LIN {X 0,Y 361.915,Z 594.733,A -85,B 0,C 180,E1 -13475.323,E2 -13475.323} C_VEL
LIN {X 0,Y 360.28,Z 612.656,A -85,B 0,C 180,E1 -13478.546,E2 -13478.546} C_VEL
LIN {X 0,Y 358.832,Z 632.276,A -85,B 0,C 180,E1 -13482.004,E2 -13482.004} C_VEL
LIN {X 0,Y 361.379,Z 647.06,A -85,B 0,C 180,E1 -13482.737,E2 -13482.737} C_VEL
LIN {X 0,Y 361.862,Z 654.515,A -85,B 0,C 180,E1 -13483.025,E2 -13483.025} C_VEL
LIN {X 0,Y 359.915,Z 705.535,A -85,B 0,C 180,E1 -13484.534,E2 -13484.534} C_VEL
LIN {X 0,Y 359.371,Z 715.25,A -85,B 0,C 180,E1 -13484.982,E2 -13484.982} C_VEL
LIN {X 0,Y 358.665,Z 725.972,A -85,B 0,C 180,E1 -13485.677,E2 -13485.677} C_VEL
LIN {X 0,Y 357.824,Z 735.392,A -85,B 0,C 180,E1 -13486.512,E2 -13486.512} C_VEL
LIN {X 0,Y 357.037,Z 744.121,A -85,B 0,C 180,E1 -13487.495,E2 -13487.495} C_VEL
LIN {X 0,Y 356.198,Z 752.116,A -85,B 0,C 180,E1 -13488.621,E2 -13488.621} C_VEL
LIN {X 0,Y 355.444,Z 758.493,A -85,B 0,C 180,E1 -13489.75,E2 -13489.75} C_VEL
LIN {X 0,Y 354.734,Z 764.94,A -85,B 0,C 180,E1 -13491.168,E2 -13491.168} C_VEL
LIN {X 0,Y 354.161,Z 770.791,A -85,B 0,C 180,E1 -13492.846,E2 -13492.846} C_VEL
LIN {X 0,Y 353.842,Z 774.432,A -85,B 0,C 180,E1 -13494.301,E2 -13494.301} C_VEL
LIN {X 0,Y 353.51,Z 776.577,A -85,B 0,C 180,E1 -13495.439,E2 -13495.439} C_VEL
LIN {X 0,Y 353.317,Z 778.1,A -85,B 0,C 180,E1 -13496.579,E2 -13496.579} C_VEL
LIN {X 0,Y 353.22,Z 779.024,A -85,B 0,C 180,E1 -13497.719,E2 -13497.719} C_VEL
LIN {X 0,Y 353.166,Z 779.339,A -85,B 0,C 180,E1 -13498.86,E2 -13498.86} C_VEL
LIN {X 0,Y 353.174,Z 779.042,A -85,B 0,C 180,E1 -13500,E2 -13500} C_VEL
LIN {X 0,Y 353.159,Z 778.151,A -85,B 0,C 180,E1 -13501.14,E2 -13501.14} C_VEL
LIN {X 0,Y 353.221,Z 775.737,A -85,B 0,C 180,E1 -13502.851,E2 -13502.851} C_VEL
LIN {X 0,Y 353.366,Z 773.306,A -85,B 0,C 180,E1 -13503.992,E2 -13503.992} C_VEL
LIN {X 0,Y 353.437,Z 770.155,A -85,B 0,C 180,E1 -13505.134,E2 -13505.134} C_VEL
LIN {X 0,Y 353.588,Z 765.013,A -85,B 0,C 180,E1 -13506.57,E2 -13506.57} C_VEL
LIN {X 0,Y 353.957,Z 758.522,A -85,B 0,C 180,E1 -13507.989,E2 -13507.989} C_VEL
LIN {X 0,Y 354.384,Z 750.124,A -85,B 0,C 180,E1 -13509.417,E2 -13509.417} C_VEL
LIN {X 0,Y 354.768,Z 742.674,A -85,B 0,C 180,E1 -13510.415,E2 -13510.415} C_VEL
LIN {X 0,Y 355.307,Z 733.469,A -85,B 0,C 180,E1 -13511.408,E2 -13511.408} C_VEL
LIN {X 0,Y 355.737,Z 722.981,A -85,B 0,C 180,E1 -13512.262,E2 -13512.262} C_VEL
LIN {X 0,Y 356.026,Z 713.566,A -85,B 0,C 180,E1 -13512.831,E2 -13512.831} C_VEL
LIN {X 0,Y 356.368,Z 702.776,A -85,B 0,C 180,E1 -13513.29,E2 -13513.29} C_VEL
LIN {X 0,Y 357.205,Z 650.23,A -85,B 0,C 180,E1 -13514.684,E2 -13514.684} C_VEL
LIN {X 0,Y 355.644,Z 631.764,A -85,B 0,C 180,E1 -13515.249,E2 -13515.249} C_VEL
LIN {X 0,Y 356.547,Z 612.473,A -85,B 0,C 180,E1 -13518.58,E2 -13518.58} C_VEL
LIN {X 0,Y 357.724,Z 591.341,A -85,B 0,C 180,E1 -13522.266,E2 -13522.266} C_VEL
LIN {X 0,Y 359.197,Z 567.38,A -85,B 0,C 180,E1 -13526.454,E2 -13526.454} C_VEL
LIN {X 0,Y 359.427,Z 562.274,A -85,B 0,C 180,E1 -13527.355,E2 -13527.355} C_VEL
LIN {X 0,Y 356.238,Z 546.772,A -85,B 0,C 180,E1 -13530.304,E2 -13530.304} C_VEL
LIN {X 0,Y 354.906,Z 540.412,A -85,B 0,C 180,E1 -13531.563,E2 -13531.563} C_VEL
LIN {X 0,Y 354.817,Z 540.288,A -85,B 0,C 180,E1 -13535.059,E2 -13535.059} C_VEL
LIN {X 0,Y 354.811,Z 540.288,A -85,B 0,C 180,E1 -13537.882,E2 -13537.882} C_VEL
LIN {X 0,Y 354.792,Z 540.268,A -85,B 0,C 180,E1 -13541.171,E2 -13541.171} C_VEL
LIN {X 0,Y 354.795,Z 540.267,A -85,B 0,C 180,E1 -13544.51,E2 -13544.51} C_VEL
LIN {X 0,Y 354.805,Z 540.287,A -85,B 0,C 180,E1 -13547.663,E2 -13547.663} C_VEL
LIN {X 0,Y 354.82,Z 540.262,A -85,B 0,C 180,E1 -13550.666,E2 -13550.666} C_VEL
LIN {X 0,Y 354.826,Z 540.285,A -85,B 0,C 180,E1 -13554.3,E2 -13554.3} C_VEL
LIN {X 0,Y 354.791,Z 540.29,A -85,B 0,C 180,E1 -13557.666,E2 -13557.666} C_VEL
LIN {X 0,Y 354.833,Z 540.286,A -85,B 0,C 180,E1 -13560.632,E2 -13560.632} C_VEL
LIN {X 0,Y 354.938,Z 540.423,A -85,B 0,C 180,E1 -13563.859,E2 -13563.859} C_VEL
LIN {X 0,Y 356.824,Z 549.95,A -85,B 0,C 180,E1 -13566.8,E2 -13566.8} C_VEL
LIN {X 0,Y 357.319,Z 552.539,A -85,B 0,C 180,E1 -13567.484,E2 -13567.484} C_VEL
LIN {X 0,Y 360.175,Z 560.697,A -85,B 0,C 180,E1 -13567.88,E2 -13567.88} C_VEL
LIN {X 0,Y 363.96,Z 579.582,A -85,B 0,C 180,E1 -13568.519,E2 -13568.519} C_VEL
LIN {X 0,Y 362.52,Z 658.642,A -85,B 0,C 180,E1 -13570.093,E2 -13570.093} C_VEL
LIN {X 0,Y 361.977,Z 672.088,A -85,B 0,C 180,E1 -13570.579,E2 -13570.579} C_VEL
LIN {X 0,Y 361.219,Z 684.867,A -85,B 0,C 180,E1 -13571.274,E2 -13571.274} C_VEL
LIN {X 0,Y 360.317,Z 696.201,A -85,B 0,C 180,E1 -13572.108,E2 -13572.108} C_VEL
LIN {X 0,Y 359.181,Z 707.773,A -85,B 0,C 180,E1 -13573.215,E2 -13573.215} C_VEL
LIN {X 0,Y 358.249,Z 718.307,A -85,B 0,C 180,E1 -13574.496,E2 -13574.496} C_VEL
LIN {X 0,Y 357.21,Z 726.851,A -85,B 0,C 180,E1 -13575.762,E2 -13575.762} C_VEL
LIN {X 0,Y 356.22,Z 734.721,A -85,B 0,C 180,E1 -13577.175,E2 -13577.175} C_VEL
LIN {X 0,Y 355.29,Z 742.409,A -85,B 0,C 180,E1 -13578.879,E2 -13578.879} C_VEL
LIN {X 0,Y 354.406,Z 749.468,A -85,B 0,C 180,E1 -13580.871,E2 -13580.871} C_VEL
LIN {X 0,Y 353.946,Z 754.166,A -85,B 0,C 180,E1 -13582.583,E2 -13582.583} C_VEL
LIN {X 0,Y 353.676,Z 757.756,A -85,B 0,C 180,E1 -13584.297,E2 -13584.297} C_VEL
LIN {X 0,Y 353.497,Z 759.613,A -85,B 0,C 180,E1 -13585.438,E2 -13585.438} C_VEL
LIN {X 0,Y 353.34,Z 761.013,A -85,B 0,C 180,E1 -13586.578,E2 -13586.578} C_VEL
LIN {X 0,Y 353.256,Z 762.621,A -85,B 0,C 180,E1 -13588.859,E2 -13588.859} C_VEL
LIN {X 0,Y 353.265,Z 762.853,A -85,B 0,C 180,E1 -13589.999,E2 -13589.999} C_VEL
LIN {X 0,Y 353.256,Z 762.665,A -85,B 0,C 180,E1 -13591.139,E2 -13591.139} C_VEL
LIN {X 0,Y 353.334,Z 761.117,A -85,B 0,C 180,E1 -13593.42,E2 -13593.42} C_VEL
LIN {X 0,Y 353.49,Z 759.761,A -85,B 0,C 180,E1 -13594.56,E2 -13594.56} C_VEL
LIN {X 0,Y 353.814,Z 756.019,A -85,B 0,C 180,E1 -13596.695,E2 -13596.695} C_VEL
LIN {X 0,Y 354.2,Z 751.45,A -85,B 0,C 180,E1 -13598.557,E2 -13598.557} C_VEL
LIN {X 0,Y 355.015,Z 745.015,A -85,B 0,C 180,E1 -13600.55,E2 -13600.55} C_VEL
LIN {X 0,Y 355.811,Z 737.943,A -85,B 0,C 180,E1 -13602.258,E2 -13602.258} C_VEL
LIN {X 0,Y 356.917,Z 729.128,A -85,B 0,C 180,E1 -13603.957,E2 -13603.957} C_VEL
LIN {X 0,Y 358.056,Z 720.077,A -85,B 0,C 180,E1 -13605.365,E2 -13605.365} C_VEL
LIN {X 0,Y 358.248,Z 718.084,A -85,B 0,C 180,E1 -13605.637,E2 -13605.637} C_VEL
LIN {X 0,Y 357.693,Z 714.653,A -85,B 0,C 180,E1 -13606.131,E2 -13606.131} C_VEL
LIN {X 0,Y 353.248,Z 705.711,A -85,B 0,C 180,E1 -13607.436,E2 -13607.436} C_VEL
LIN {X 0,Y 353.002,Z 702.399,A -85,B 0,C 180,E1 -13607.799,E2 -13607.799} C_VEL
LIN {X 0,Y 354.134,Z 690.557,A -85,B 0,C 180,E1 -13608.812,E2 -13608.812} C_VEL
LIN {X 0,Y 355.058,Z 678.47,A -85,B 0,C 180,E1 -13609.587,E2 -13609.587} C_VEL
LIN {X 0,Y 355.635,Z 666.212,A -85,B 0,C 180,E1 -13610.156,E2 -13610.156} C_VEL
LIN {X 0,Y 356.104,Z 654.129,A -85,B 0,C 180,E1 -13610.505,E2 -13610.505} C_VEL
LIN {X 0,Y 357.351,Z 579.83,A -85,B 0,C 180,E1 -13612.003,E2 -13612.003} C_VEL
LIN {X 0,Y 353.421,Z 561.516,A -85,B 0,C 180,E1 -13612.658,E2 -13612.658} C_VEL
LIN {X 0,Y 350.203,Z 552.682,A -85,B 0,C 180,E1 -13613.115,E2 -13613.115} C_VEL
LIN {X 0,Y 348.907,Z 546.369,A -85,B 0,C 180,E1 -13614.983,E2 -13614.983} C_VEL
LIN {X 0,Y 347.866,Z 541.204,A -85,B 0,C 180,E1 -13616.687,E2 -13616.687} C_VEL
LIN {X 0,Y 347.747,Z 541.157,A -85,B 0,C 180,E1 -13620.347,E2 -13620.347} C_VEL
LIN {X 0,Y 347.746,Z 541.17,A -85,B 0,C 180,E1 -13624.043,E2 -13624.043} C_VEL
LIN {X 0,Y 347.763,Z 541.166,A -85,B 0,C 180,E1 -13627.319,E2 -13627.319} C_VEL
LIN {X 0,Y 347.74,Z 541.16,A -85,B 0,C 180,E1 -13630.294,E2 -13630.294} C_VEL
LIN {X 0,Y 347.72,Z 541.166,A -85,B 0,C 180,E1 -13633.407,E2 -13633.407} C_VEL
LIN {X 0,Y 347.742,Z 541.163,A -85,B 0,C 180,E1 -13636.681,E2 -13636.681} C_VEL
LIN {X 0,Y 347.753,Z 541.153,A -85,B 0,C 180,E1 -13640.17,E2 -13640.17} C_VEL
LIN {X 0,Y 347.762,Z 541.151,A -85,B 0,C 180,E1 -13642.679,E2 -13642.679} C_VEL
LIN {X 0,Y 347.757,Z 541.165,A -85,B 0,C 180,E1 -13645.952,E2 -13645.952} C_VEL
LIN {X 0,Y 347.758,Z 541.169,A -85,B 0,C 180,E1 -13649.653,E2 -13649.653} C_VEL
LIN {X 0,Y 347.846,Z 541.145,A -85,B 0,C 180,E1 -13652.744,E2 -13652.744} C_VEL
LIN {X 0,Y 347.782,Z 541.159,A -85,B 0,C 180,E1 -13656.161,E2 -13656.161} C_VEL
LIN {X 0,Y 347.811,Z 541.159,A -85,B 0,C 180,E1 -13659.909,E2 -13659.909} C_VEL
LIN {X 0,Y 347.859,Z 541.147,A -85,B 0,C 180,E1 -13662.359,E2 -13662.359} C_VEL
LIN {X 0,Y 347.89,Z 541.149,A -85,B 0,C 180,E1 -13665.97,E2 -13665.97} C_VEL
LIN {X 0,Y 347.921,Z 541.135,A -85,B 0,C 180,E1 -13669.525,E2 -13669.525} C_VEL
LIN {X 0,Y 348.067,Z 541.126,A -85,B 0,C 180,E1 -13671.874,E2 -13671.874} C_VEL
LIN {X 0,Y 348.06,Z 541.126,A -85,B 0,C 180,E1 -13674.205,E2 -13674.205} C_VEL
LIN {X 0,Y 348.201,Z 541.102,A -85,B 0,C 180,E1 -13677.686,E2 -13677.686} C_VEL
LIN {X 0,Y 348.361,Z 541.091,A -85,B 0,C 180,E1 -13680,E2 -13680} C_VEL
LIN {X 0,Y 348.201,Z 541.103,A -85,B 0,C 180,E1 -13682.313,E2 -13682.313} C_VEL
LIN {X 0,Y 348.101,Z 541.122,A -85,B 0,C 180,E1 -13686.958,E2 -13686.958} C_VEL
LIN {X 0,Y 347.961,Z 541.134,A -85,B 0,C 180,E1 -13689.299,E2 -13689.299} C_VEL
LIN {X 0,Y 347.886,Z 541.148,A -85,B 0,C 180,E1 -13692.84,E2 -13692.84} C_VEL
LIN {X 0,Y 347.832,Z 541.147,A -85,B 0,C 180,E1 -13696.432,E2 -13696.432} C_VEL
LIN {X 0,Y 347.852,Z 541.153,A -85,B 0,C 180,E1 -13698.86,E2 -13698.86} C_VEL
LIN {X 0,Y 347.77,Z 541.159,A -85,B 0,C 180,E1 -13702.58,E2 -13702.58} C_VEL
LIN {X 0,Y 347.806,Z 541.16,A -85,B 0,C 180,E1 -13705.109,E2 -13705.109} C_VEL
LIN {X 0,Y 347.801,Z 541.158,A -85,B 0,C 180,E1 -13707.695,E2 -13707.695} C_VEL
LIN {X 0,Y 347.742,Z 541.163,A -85,B 0,C 180,E1 -13710.349,E2 -13710.349} C_VEL
LIN {X 0,Y 347.742,Z 541.165,A -85,B 0,C 180,E1 -13714.045,E2 -13714.045} C_VEL
LIN {X 0,Y 347.757,Z 541.148,A -85,B 0,C 180,E1 -13717.322,E2 -13717.322} C_VEL
LIN {X 0,Y 347.727,Z 541.169,A -85,B 0,C 180,E1 -13720.298,E2 -13720.298} C_VEL
LIN {X 0,Y 347.742,Z 541.158,A -85,B 0,C 180,E1 -13723.405,E2 -13723.405} C_VEL
LIN {X 0,Y 347.778,Z 541.155,A -85,B 0,C 180,E1 -13726.677,E2 -13726.677} C_VEL
LIN {X 0,Y 347.782,Z 541.157,A -85,B 0,C 180,E1 -13730.166,E2 -13730.166} C_VEL
LIN {X 0,Y 347.786,Z 541.158,A -85,B 0,C 180,E1 -13734.126,E2 -13734.126} C_VEL
LIN {X 0,Y 347.732,Z 541.104,A -85,B 0,C 180,E1 -13738.088,E2 -13738.088} C_VEL
LIN {X 0,Y 347.806,Z 541.332,A -85,B 0,C 180,E1 -13739.197,E2 -13739.197} C_VEL
LIN {X 0,Y 350.44,Z 553.084,A -85,B 0,C 180,E1 -13742.533,E2 -13742.533} C_VEL
LIN {X 0,Y 351.969,Z 561.98,A -85,B 0,C 180,E1 -13744.92,E2 -13744.92} C_VEL
LIN {X 0,Y 351.14,Z 570.572,A -85,B 0,C 180,E1 -13746.977,E2 -13746.977} C_VEL
LIN {X 0,Y 352.793,Z 579.781,A -85,B 0,C 180,E1 -13747.333,E2 -13747.333} C_VEL
LIN {X 0,Y 356.992,Z 605.545,A -85,B 0,C 180,E1 -13748.159,E2 -13748.159} C_VEL
LIN {X 0,Y 355.689,Z 678.841,A -85,B 0,C 180,E1 -13749.659,E2 -13749.659} C_VEL
LIN {X 0,Y 354.909,Z 692.03,A -85,B 0,C 180,E1 -13750.141,E2 -13750.141} C_VEL
LIN {X 0,Y 354.07,Z 704.157,A -85,B 0,C 180,E1 -13750.808,E2 -13750.808} C_VEL
LIN {X 0,Y 352.939,Z 716.406,A -85,B 0,C 180,E1 -13751.723,E2 -13751.723} C_VEL
LIN {X 0,Y 351.697,Z 727.988,A -85,B 0,C 180,E1 -13752.859,E2 -13752.859} C_VEL
LIN {X 0,Y 350.453,Z 738.96,A -85,B 0,C 180,E1 -13754.22,E2 -13754.22} C_VEL
LIN {X 0,Y 349.342,Z 748.628,A -85,B 0,C 180,E1 -13755.734,E2 -13755.734} C_VEL
LIN {X 0,Y 348.199,Z 757.561,A -85,B 0,C 180,E1 -13757.47,E2 -13757.47} C_VEL
LIN {X 0,Y 347.398,Z 764.755,A -85,B 0,C 180,E1 -13759.216,E2 -13759.216} C_VEL
LIN {X 0,Y 346.719,Z 771.306,A -85,B 0,C 180,E1 -13761.257,E2 -13761.257} C_VEL
LIN {X 0,Y 346.343,Z 775.644,A -85,B 0,C 180,E1 -13763.008,E2 -13763.008} C_VEL
LIN {X 0,Y 346.2,Z 777.944,A -85,B 0,C 180,E1 -13764.175,E2 -13764.175} C_VEL
LIN {X 0,Y 346.175,Z 779.809,A -85,B 0,C 180,E1 -13765.343,E2 -13765.343} C_VEL
LIN {X 0,Y 346.147,Z 781.205,A -85,B 0,C 180,E1 -13766.509,E2 -13766.509} C_VEL
LIN {X 0,Y 346.123,Z 784.253,A -85,B 0,C 180,E1 -13770.001,E2 -13770.001} C_VEL
LIN {X 0,Y 346.069,Z 784.599,A -85,B 0,C 180,E1 -13771.165,E2 -13771.165} C_VEL
LIN {X 0,Y 346.081,Z 784.32,A -85,B 0,C 180,E1 -13772.329,E2 -13772.329} C_VEL
LIN {X 0,Y 346.154,Z 783.447,A -85,B 0,C 180,E1 -13773.493,E2 -13773.493} C_VEL
LIN {X 0,Y 346.257,Z 781.07,A -85,B 0,C 180,E1 -13775.242,E2 -13775.242} C_VEL
LIN {X 0,Y 346.431,Z 777.124,A -85,B 0,C 180,E1 -13776.992,E2 -13776.992} C_VEL
LIN {X 0,Y 346.615,Z 773.662,A -85,B 0,C 180,E1 -13778.161,E2 -13778.161} C_VEL
LIN {X 0,Y 347.574,Z 762.458,A -85,B 0,C 180,E1 -13781.371,E2 -13781.371} C_VEL
LIN {X 0,Y 348.549,Z 754.751,A -85,B 0,C 180,E1 -13783.112,E2 -13783.112} C_VEL
LIN {X 0,Y 349.714,Z 745.072,A -85,B 0,C 180,E1 -13784.847,E2 -13784.847} C_VEL
LIN {X 0,Y 350.835,Z 735.09,A -85,B 0,C 180,E1 -13786.288,E2 -13786.288} C_VEL
LIN {X 0,Y 352.096,Z 723.812,A -85,B 0,C 180,E1 -13787.573,E2 -13787.573} C_VEL
LIN {X 0,Y 353.272,Z 712.771,A -85,B 0,C 180,E1 -13788.561,E2 -13788.561} C_VEL
LIN {X 0,Y 354.315,Z 700.533,A -85,B 0,C 180,E1 -13789.406,E2 -13789.406} C_VEL
LIN {X 0,Y 355.211,Z 687.646,A -85,B 0,C 180,E1 -13790.032,E2 -13790.032} C_VEL
LIN {X 0,Y 355.763,Z 673.928,A -85,B 0,C 180,E1 -13790.452,E2 -13790.452} C_VEL
LIN {X 0,Y 356.868,Z 604.856,A -85,B 0,C 180,E1 -13791.849,E2 -13791.849} C_VEL
LIN {X 0,Y 353.3,Z 582.279,A -85,B 0,C 180,E1 -13792.598,E2 -13792.598} C_VEL
LIN {X 0,Y 353.345,Z 575.714,A -85,B 0,C 180,E1 -13793.269,E2 -13793.269} C_VEL
LIN {X 0,Y 352.557,Z 568.23,A -85,B 0,C 180,E1 -13794.231,E2 -13794.231} C_VEL
LIN {X 0,Y 352.055,Z 562.274,A -85,B 0,C 180,E1 -13795.073,E2 -13795.073} C_VEL
LIN {X 0,Y 350.889,Z 555.527,A -85,B 0,C 180,E1 -13796.787,E2 -13796.787} C_VEL
LIN {X 0,Y 348.952,Z 546.205,A -85,B 0,C 180,E1 -13799.368,E2 -13799.368} C_VEL
LIN {X 0,Y 347.804,Z 541.253,A -85,B 0,C 180,E1 -13800.848,E2 -13800.848} C_VEL
LIN {X 0,Y 347.748,Z 541.171,A -85,B 0,C 180,E1 -13804.464,E2 -13804.464} C_VEL
LIN {X 0,Y 347.777,Z 541.167,A -85,B 0,C 180,E1 -13807.989,E2 -13807.989} C_VEL
LIN {X 0,Y 347.755,Z 541.169,A -85,B 0,C 180,E1 -13811.831,E2 -13811.831} C_VEL
LIN {X 0,Y 347.71,Z 541.173,A -85,B 0,C 180,E1 -13815.027,E2 -13815.027} C_VEL
LIN {X 0,Y 347.754,Z 541.168,A -85,B 0,C 180,E1 -13818.398,E2 -13818.398} C_VEL
LIN {X 0,Y 347.821,Z 541.434,A -85,B 0,C 180,E1 -13820.846,E2 -13820.846} C_VEL
LIN {X 0,Y 349.991,Z 546.723,A -85,B 0,C 180,E1 -13822.957,E2 -13822.957} C_VEL
LIN {X 0,Y 352.71,Z 553.567,A -85,B 0,C 180,E1 -13825.28,E2 -13825.28} C_VEL
LIN {X 0,Y 355.393,Z 562,A -85,B 0,C 180,E1 -13827.728,E2 -13827.728} C_VEL
LIN {X 0,Y 357.118,Z 569.16,A -85,B 0,C 180,E1 -13829.556,E2 -13829.556} C_VEL
LIN {X 0,Y 357.945,Z 575.077,A -85,B 0,C 180,E1 -13830.925,E2 -13830.925} C_VEL
LIN {X 0,Y 355.927,Z 592.958,A -85,B 0,C 180,E1 -13834.253,E2 -13834.253} C_VEL
LIN {X 0,Y 353.975,Z 612.503,A -85,B 0,C 180,E1 -13837.837,E2 -13837.837} C_VEL
LIN {X 0,Y 352.348,Z 632.152,A -85,B 0,C 180,E1 -13841.389,E2 -13841.389} C_VEL
LIN {X 0,Y 354.995,Z 647.631,A -85,B 0,C 180,E1 -13842.213,E2 -13842.213} C_VEL
LIN {X 0,Y 355.568,Z 654.786,A -85,B 0,C 180,E1 -13842.508,E2 -13842.508} C_VEL
LIN {X 0,Y 353.443,Z 705.58,A -85,B 0,C 180,E1 -13844.059,E2 -13844.059} C_VEL
LIN {X 0,Y 352.848,Z 715.786,A -85,B 0,C 180,E1 -13844.55,E2 -13844.55} C_VEL
LIN {X 0,Y 352.063,Z 726.264,A -85,B 0,C 180,E1 -13845.255,E2 -13845.255} C_VEL
LIN {X 0,Y 351.177,Z 735.596,A -85,B 0,C 180,E1 -13846.104,E2 -13846.104} C_VEL
LIN {X 0,Y 350.334,Z 744.318,A -85,B 0,C 180,E1 -13847.104,E2 -13847.104} C_VEL
LIN {X 0,Y 349.31,Z 753.123,A -85,B 0,C 180,E1 -13848.393,E2 -13848.393} C_VEL
LIN {X 0,Y 348.519,Z 759.359,A -85,B 0,C 180,E1 -13849.544,E2 -13849.544} C_VEL
LIN {X 0,Y 347.907,Z 764.489,A -85,B 0,C 180,E1 -13850.7,E2 -13850.7} C_VEL
LIN {X 0,Y 347.314,Z 769.751,A -85,B 0,C 180,E1 -13852.179,E2 -13852.179} C_VEL
LIN {X 0,Y 346.981,Z 773.598,A -85,B 0,C 180,E1 -13853.604,E2 -13853.604} C_VEL
LIN {X 0,Y 346.459,Z 776.857,A -85,B 0,C 180,E1 -13855.346,E2 -13855.346} C_VEL
LIN {X 0,Y 346.245,Z 778.294,A -85,B 0,C 180,E1 -13856.509,E2 -13856.509} C_VEL
LIN {X 0,Y 346.131,Z 779.14,A -85,B 0,C 180,E1 -13857.673,E2 -13857.673} C_VEL
LIN {X 0,Y 346.069,Z 779.396,A -85,B 0,C 180,E1 -13858.836,E2 -13858.836} C_VEL
LIN {X 0,Y 346.075,Z 779.038,A -85,B 0,C 180,E1 -13860,E2 -13860} C_VEL
LIN {X 0,Y 346.062,Z 778.065,A -85,B 0,C 180,E1 -13861.164,E2 -13861.164} C_VEL
LIN {X 0,Y 346.142,Z 775.463,A -85,B 0,C 180,E1 -13862.91,E2 -13862.91} C_VEL
LIN {X 0,Y 346.327,Z 771.383,A -85,B 0,C 180,E1 -13864.656,E2 -13864.656} C_VEL
LIN {X 0,Y 346.451,Z 766.163,A -85,B 0,C 180,E1 -13866.274,E2 -13866.274} C_VEL
LIN {X 0,Y 346.772,Z 760.656,A -85,B 0,C 180,E1 -13867.57,E2 -13867.57} C_VEL
LIN {X 0,Y 347.053,Z 754.557,A -85,B 0,C 180,E1 -13868.736,E2 -13868.736} C_VEL
LIN {X 0,Y 347.516,Z 747.094,A -85,B 0,C 180,E1 -13869.898,E2 -13869.898} C_VEL
LIN {X 0,Y 347.944,Z 737.609,A -85,B 0,C 180,E1 -13871.063,E2 -13871.063} C_VEL
LIN {X 0,Y 348.344,Z 730.147,A -85,B 0,C 180,E1 -13871.787,E2 -13871.787} C_VEL
LIN {X 0,Y 348.734,Z 720.716,A -85,B 0,C 180,E1 -13872.512,E2 -13872.512} C_VEL
LIN {X 0,Y 349.065,Z 709.842,A -85,B 0,C 180,E1 -13873.129,E2 -13873.129} C_VEL
LIN {X 0,Y 349.317,Z 698.696,A -85,B 0,C 180,E1 -13873.526,E2 -13873.526} C_VEL
LIN {X 0,Y 350.173,Z 650.419,A -85,B 0,C 180,E1 -13874.836,E2 -13874.836} C_VEL
LIN {X 0,Y 348.579,Z 631.804,A -85,B 0,C 180,E1 -13875.42,E2 -13875.42} C_VEL
LIN {X 0,Y 349.497,Z 614.378,A -85,B 0,C 180,E1 -13878.465,E2 -13878.465} C_VEL
LIN {X 0,Y 350.718,Z 592.221,A -85,B 0,C 180,E1 -13882.38,E2 -13882.38} C_VEL
LIN {X 0,Y 352.133,Z 569.733,A -85,B 0,C 180,E1 -13886.364,E2 -13886.364} C_VEL
LIN {X 0,Y 352.366,Z 562.799,A -85,B 0,C 180,E1 -13887.606,E2 -13887.606} C_VEL
LIN {X 0,Y 348.783,Z 545.615,A -85,B 0,C 180,E1 -13890.919,E2 -13890.919} C_VEL
LIN {X 0,Y 347.831,Z 541.279,A -85,B 0,C 180,E1 -13891.824,E2 -13891.824} C_VEL
LIN {X 0,Y 347.775,Z 541.166,A -85,B 0,C 180,E1 -13896.065,E2 -13896.065} C_VEL
LIN {X 0,Y 347.757,Z 541.165,A -85,B 0,C 180,E1 -13898.792,E2 -13898.792} C_VEL
LIN {X 0,Y 347.755,Z 541.134,A -85,B 0,C 180,E1 -13901.83,E2 -13901.83} C_VEL
LIN {X 0,Y 347.773,Z 541.149,A -85,B 0,C 180,E1 -13905.016,E2 -13905.016} C_VEL
LIN {X 0,Y 347.758,Z 541.158,A -85,B 0,C 180,E1 -13908.396,E2 -13908.396} C_VEL
LIN {X 0,Y 347.778,Z 541.153,A -85,B 0,C 180,E1 -13912.011,E2 -13912.011} C_VEL
LIN {X 0,Y 347.749,Z 541.156,A -85,B 0,C 180,E1 -13915.536,E2 -13915.536} C_VEL
LIN {X 0,Y 347.765,Z 541.165,A -85,B 0,C 180,E1 -13919.653,E2 -13919.653} C_VEL
LIN {X 0,Y 347.898,Z 541.272,A -85,B 0,C 180,E1 -13923.48,E2 -13923.48} C_VEL
LIN {X 0,Y 349.965,Z 551.705,A -85,B 0,C 180,E1 -13926.765,E2 -13926.765} C_VEL
LIN {X 0,Y 350.215,Z 552.95,A -85,B 0,C 180,E1 -13927.018,E2 -13927.018} C_VEL
LIN {X 0,Y 353.926,Z 563.384,A -85,B 0,C 180,E1 -13927.522,E2 -13927.522} C_VEL
LIN {X 0,Y 357.365,Z 580.665,A -85,B 0,C 180,E1 -13928.12,E2 -13928.12} C_VEL
LIN {X 0,Y 355.876,Z 658.864,A -85,B 0,C 180,E1 -13929.705,E2 -13929.705} C_VEL
LIN {X 0,Y 355.298,Z 672.303,A -85,B 0,C 180,E1 -13930.199,E2 -13930.199} C_VEL
LIN {X 0,Y 354.52,Z 685.079,A -85,B 0,C 180,E1 -13930.907,E2 -13930.907} C_VEL
LIN {X 0,Y 353.585,Z 696.411,A -85,B 0,C 180,E1 -13931.756,E2 -13931.756} C_VEL
LIN {X 0,Y 352.511,Z 706.905,A -85,B 0,C 180,E1 -13932.763,E2 -13932.763} C_VEL
LIN {X 0,Y 351.509,Z 717.451,A -85,B 0,C 180,E1 -13934.042,E2 -13934.042} C_VEL
LIN {X 0,Y 350.339,Z 727.058,A -85,B 0,C 180,E1 -13935.477,E2 -13935.477} C_VEL
LIN {X 0,Y 349.282,Z 734.929,A -85,B 0,C 180,E1 -13936.916,E2 -13936.916} C_VEL
LIN {X 0,Y 348.321,Z 742.616,A -85,B 0,C 180,E1 -13938.654,E2 -13938.654} C_VEL
LIN {X 0,Y 347.656,Z 747.864,A -85,B 0,C 180,E1 -13940.105,E2 -13940.105} C_VEL
LIN {X 0,Y 347.019,Z 752.957,A -85,B 0,C 180,E1 -13941.849,E2 -13941.849} C_VEL
LIN {X 0,Y 346.728,Z 756.326,A -85,B 0,C 180,E1 -13943.32,E2 -13943.32} C_VEL
LIN {X 0,Y 346.439,Z 759.818,A -85,B 0,C 180,E1 -13945.345,E2 -13945.345} C_VEL
LIN {X 0,Y 346.264,Z 761.218,A -85,B 0,C 180,E1 -13946.508,E2 -13946.508} C_VEL
LIN {X 0,Y 346.16,Z 762.826,A -85,B 0,C 180,E1 -13948.836,E2 -13948.836} C_VEL
LIN {X 0,Y 346.168,Z 763.058,A -85,B 0,C 180,E1 -13949.999,E2 -13949.999} C_VEL
LIN {X 0,Y 346.159,Z 762.869,A -85,B 0,C 180,E1 -13951.162,E2 -13951.162} C_VEL
LIN {X 0,Y 346.259,Z 761.321,A -85,B 0,C 180,E1 -13953.49,E2 -13953.49} C_VEL
LIN {X 0,Y 346.432,Z 759.964,A -85,B 0,C 180,E1 -13954.653,E2 -13954.653} C_VEL
LIN {X 0,Y 346.727,Z 756.547,A -85,B 0,C 180,E1 -13956.679,E2 -13956.679} C_VEL
LIN {X 0,Y 347.175,Z 751.654,A -85,B 0,C 180,E1 -13958.732,E2 -13958.732} C_VEL
LIN {X 0,Y 348.004,Z 745.219,A -85,B 0,C 180,E1 -13960.765,E2 -13960.765} C_VEL
LIN {X 0,Y 348.861,Z 738.146,A -85,B 0,C 180,E1 -13962.506,E2 -13962.506} C_VEL
LIN {X 0,Y 350.045,Z 729.329,A -85,B 0,C 180,E1 -13964.237,E2 -13964.237} C_VEL
LIN {X 0,Y 351.213,Z 720.288,A -85,B 0,C 180,E1 -13965.67,E2 -13965.67} C_VEL
LIN {X 0,Y 352.302,Z 709.234,A -85,B 0,C 180,E1 -13967.081,E2 -13967.081} C_VEL
LIN {X 0,Y 353.002,Z 702.399,A -85,B 0,C 180,E1 -13967.799,E2 -13967.799} C_VEL
LIN {X 0,Y 352.983,Z 697.369,A -85,B 0,C 180,E1 -13968.302,E2 -13968.302} C_VEL
LIN {X 0,Y 351.028,Z 689.052,A -85,B 0,C 180,E1 -13969.125,E2 -13969.125} C_VEL
LIN {X 0,Y 348.89,Z 680.413,A -85,B 0,C 180,E1 -13969.847,E2 -13969.847} C_VEL
LIN {X 0,Y 348.576,Z 674.878,A -85,B 0,C 180,E1 -13970.184,E2 -13970.184} C_VEL
LIN {X 0,Y 349.199,Z 663.426,A -85,B 0,C 180,E1 -13970.66,E2 -13970.66} C_VEL
LIN {X 0,Y 349.622,Z 645.492,A -85,B 0,C 180,E1 -13971.096,E2 -13971.096} C_VEL
LIN {X 0,Y 350.73,Z 580.722,A -85,B 0,C 180,E1 -13972.426,E2 -13972.426} C_VEL
LIN {X 0,Y 347.06,Z 563.542,A -85,B 0,C 180,E1 -13973.057,E2 -13973.057} C_VEL
LIN {X 0,Y 343.049,Z 552.944,A -85,B 0,C 180,E1 -13973.62,E2 -13973.62} C_VEL
LIN {X 0,Y 341.508,Z 545.362,A -85,B 0,C 180,E1 -13975.931,E2 -13975.931} C_VEL
LIN {X 0,Y 340.834,Z 542.049,A -85,B 0,C 180,E1 -13977.111,E2 -13977.111} C_VEL
LIN {X 0,Y 340.696,Z 542.044,A -85,B 0,C 180,E1 -13981.043,E2 -13981.043} C_VEL
LIN {X 0,Y 340.716,Z 542.04,A -85,B 0,C 180,E1 -13985.277,E2 -13985.277} C_VEL
LIN {X 0,Y 340.71,Z 542.043,A -85,B 0,C 180,E1 -13988.386,E2 -13988.386} C_VEL
LIN {X 0,Y 340.699,Z 542.046,A -85,B 0,C 180,E1 -13992.045,E2 -13992.045} C_VEL
LIN {X 0,Y 340.663,Z 542.045,A -85,B 0,C 180,E1 -13996.223,E2 -13996.223} C_VEL
LIN {X 0,Y 340.7,Z 542.044,A -85,B 0,C 180,E1 -13998.692,E2 -13998.692} C_VEL
LIN {X 0,Y 340.736,Z 542.019,A -85,B 0,C 180,E1 -14001.773,E2 -14001.773} C_VEL
LIN {X 0,Y 340.727,Z 542.044,A -85,B 0,C 180,E1 -14005.592,E2 -14005.592} C_VEL
LIN {X 0,Y 340.757,Z 542.038,A -85,B 0,C 180,E1 -14010.021,E2 -14010.021} C_VEL
LIN {X 0,Y 340.799,Z 542.024,A -85,B 0,C 180,E1 -14013.019,E2 -14013.019} C_VEL
LIN {X 0,Y 340.722,Z 542.039,A -85,B 0,C 180,E1 -14016.927,E2 -14016.927} C_VEL
LIN {X 0,Y 340.788,Z 542.032,A -85,B 0,C 180,E1 -14020.733,E2 -14020.733} C_VEL
LIN {X 0,Y 340.779,Z 542.026,A -85,B 0,C 180,E1 -14023.218,E2 -14023.218} C_VEL
LIN {X 0,Y 340.837,Z 542.027,A -85,B 0,C 180,E1 -14026.89,E2 -14026.89} C_VEL
LIN {X 0,Y 340.921,Z 542.004,A -85,B 0,C 180,E1 -14030.507,E2 -14030.507} C_VEL
LIN {X 0,Y 341.068,Z 541.997,A -85,B 0,C 180,E1 -14032.898,E2 -14032.898} C_VEL
LIN {X 0,Y 341.163,Z 541.977,A -85,B 0,C 180,E1 -14037.639,E2 -14037.639} C_VEL
LIN {X 0,Y 341.31,Z 541.97,A -85,B 0,C 180,E1 -14040,E2 -14040} C_VEL
LIN {X 0,Y 341.163,Z 541.979,A -85,B 0,C 180,E1 -14042.361,E2 -14042.361} C_VEL
LIN {X 0,Y 341.07,Z 541.999,A -85,B 0,C 180,E1 -14047.102,E2 -14047.102} C_VEL
LIN {X 0,Y 340.866,Z 542.013,A -85,B 0,C 180,E1 -14050.694,E2 -14050.694} C_VEL
LIN {X 0,Y 340.855,Z 542.022,A -85,B 0,C 180,E1 -14054.325,E2 -14054.325} C_VEL
LIN {X 0,Y 340.831,Z 542.027,A -85,B 0,C 180,E1 -14058.468,E2 -14058.468} C_VEL
LIN {X 0,Y 340.746,Z 542.033,A -85,B 0,C 180,E1 -14061.857,E2 -14061.857} C_VEL
LIN {X 0,Y 340.765,Z 542.034,A -85,B 0,C 180,E1 -14065.665,E2 -14065.665} C_VEL
LIN {X 0,Y 340.721,Z 542.042,A -85,B 0,C 180,E1 -14068.321,E2 -14068.321} C_VEL
LIN {X 0,Y 340.691,Z 542.041,A -85,B 0,C 180,E1 -14071.045,E2 -14071.045} C_VEL
LIN {X 0,Y 340.712,Z 542.032,A -85,B 0,C 180,E1 -14075.28,E2 -14075.28} C_VEL
LIN {X 0,Y 340.705,Z 542.042,A -85,B 0,C 180,E1 -14078.387,E2 -14078.387} C_VEL
LIN {X 0,Y 340.696,Z 542.032,A -85,B 0,C 180,E1 -14082.047,E2 -14082.047} C_VEL
LIN {X 0,Y 340.731,Z 542.043,A -85,B 0,C 180,E1 -14085.471,E2 -14085.471} C_VEL
LIN {X 0,Y 340.721,Z 542.043,A -85,B 0,C 180,E1 -14088.697,E2 -14088.697} C_VEL
LIN {X 0,Y 340.735,Z 542.013,A -85,B 0,C 180,E1 -14091.775,E2 -14091.775} C_VEL
LIN {X 0,Y 340.72,Z 542.037,A -85,B 0,C 180,E1 -14095.596,E2 -14095.596} C_VEL
LIN {X 0,Y 340.735,Z 542.067,A -85,B 0,C 180,E1 -14098.702,E2 -14098.702} C_VEL
LIN {X 0,Y 343.178,Z 552.874,A -85,B 0,C 180,E1 -14101.901,E2 -14101.901} C_VEL
LIN {X 0,Y 345.004,Z 562.916,A -85,B 0,C 180,E1 -14104.674,E2 -14104.674} C_VEL
LIN {X 0,Y 344.445,Z 569.181,A -85,B 0,C 180,E1 -14106.252,E2 -14106.252} C_VEL
LIN {X 0,Y 344.392,Z 570.812,A -85,B 0,C 180,E1 -14106.533,E2 -14106.533} C_VEL
LIN {X 0,Y 349.428,Z 599.924,A -85,B 0,C 180,E1 -14107.543,E2 -14107.543} C_VEL
LIN {X 0,Y 350.388,Z 608.082,A -85,B 0,C 180,E1 -14107.784,E2 -14107.784} C_VEL
LIN {X 0,Y 349.044,Z 678.649,A -85,B 0,C 180,E1 -14109.254,E2 -14109.254} C_VEL
LIN {X 0,Y 348.247,Z 691.834,A -85,B 0,C 180,E1 -14109.744,E2 -14109.744} C_VEL
LIN {X 0,Y 347.369,Z 703.959,A -85,B 0,C 180,E1 -14110.423,E2 -14110.423} C_VEL
LIN {X 0,Y 346.199,Z 716.206,A -85,B 0,C 180,E1 -14111.354,E2 -14111.354} C_VEL
LIN {X 0,Y 344.91,Z 727.787,A -85,B 0,C 180,E1 -14112.511,E2 -14112.511} C_VEL
LIN {X 0,Y 343.683,Z 737.768,A -85,B 0,C 180,E1 -14113.76,E2 -14113.76} C_VEL
LIN {X 0,Y 342.61,Z 746.748,A -85,B 0,C 180,E1 -14115.144,E2 -14115.144} C_VEL
LIN {X 0,Y 341.623,Z 754.621,A -85,B 0,C 180,E1 -14116.619,E2 -14116.619} C_VEL
LIN {X 0,Y 340.578,Z 762.31,A -85,B 0,C 180,E1 -14118.394,E2 -14118.394} C_VEL
LIN {X 0,Y 340.035,Z 767.584,A -85,B 0,C 180,E1 -14119.883,E2 -14119.883} C_VEL
LIN {X 0,Y 339.53,Z 772.693,A -85,B 0,C 180,E1 -14121.67,E2 -14121.67} C_VEL
LIN {X 0,Y 339.175,Z 776.666,A -85,B 0,C 180,E1 -14123.457,E2 -14123.457} C_VEL
LIN {X 0,Y 339.076,Z 779.604,A -85,B 0,C 180,E1 -14125.245,E2 -14125.245} C_VEL
LIN {X 0,Y 339.071,Z 781.001,A -85,B 0,C 180,E1 -14126.436,E2 -14126.436} C_VEL
LIN {X 0,Y 339.025,Z 784.082,A -85,B 0,C 180,E1 -14130.001,E2 -14130.001} C_VEL
LIN {X 0,Y 338.974,Z 784.495,A -85,B 0,C 180,E1 -14131.189,E2 -14131.189} C_VEL
LIN {X 0,Y 338.996,Z 784.308,A -85,B 0,C 180,E1 -14132.377,E2 -14132.377} C_VEL
LIN {X 0,Y 339.083,Z 783.534,A -85,B 0,C 180,E1 -14133.566,E2 -14133.566} C_VEL
LIN {X 0,Y 339.174,Z 782.165,A -85,B 0,C 180,E1 -14134.755,E2 -14134.755} C_VEL
LIN {X 0,Y 339.291,Z 778.97,A -85,B 0,C 180,E1 -14136.542,E2 -14136.542} C_VEL
LIN {X 0,Y 339.61,Z 774.18,A -85,B 0,C 180,E1 -14138.33,E2 -14138.33} C_VEL
LIN {X 0,Y 339.93,Z 768.846,A -85,B 0,C 180,E1 -14139.822,E2 -14139.822} C_VEL
LIN {X 0,Y 341.062,Z 758.612,A -85,B 0,C 180,E1 -14142.497,E2 -14142.497} C_VEL
LIN {X 0,Y 342.187,Z 749.97,A -85,B 0,C 180,E1 -14144.269,E2 -14144.269} C_VEL
LIN {X 0,Y 343.301,Z 740.669,A -85,B 0,C 180,E1 -14145.808,E2 -14145.808} C_VEL
LIN {X 0,Y 344.548,Z 730.205,A -85,B 0,C 180,E1 -14147.204,E2 -14147.204} C_VEL
LIN {X 0,Y 345.832,Z 719.197,A -85,B 0,C 180,E1 -14148.361,E2 -14148.361} C_VEL
LIN {X 0,Y 347.086,Z 706.87,A -85,B 0,C 180,E1 -14149.365,E2 -14149.365} C_VEL
LIN {X 0,Y 348.003,Z 695.188,A -85,B 0,C 180,E1 -14150.08,E2 -14150.08} C_VEL
LIN {X 0,Y 348.843,Z 682.703,A -85,B 0,C 180,E1 -14150.607,E2 -14150.607} C_VEL
LIN {X 0,Y 349.29,Z 666.77,A -85,B 0,C 180,E1 -14151.003,E2 -14151.003} C_VEL
LIN {X 0,Y 350.262,Z 605.856,A -85,B 0,C 180,E1 -14152.257,E2 -14152.257} C_VEL
LIN {X 0,Y 347.594,Z 588.463,A -85,B 0,C 180,E1 -14152.831,E2 -14152.831} C_VEL
LIN {X 0,Y 347.893,Z 578.676,A -85,B 0,C 180,E1 -14153.831,E2 -14153.831} C_VEL
LIN {X 0,Y 347.302,Z 571.517,A -85,B 0,C 180,E1 -14154.797,E2 -14154.797} C_VEL
LIN {X 0,Y 346.827,Z 565.788,A -85,B 0,C 180,E1 -14155.625,E2 -14155.625} C_VEL
LIN {X 0,Y 343.781,Z 554.509,A -85,B 0,C 180,E1 -14158.048,E2 -14158.048} C_VEL
LIN {X 0,Y 341.81,Z 546.171,A -85,B 0,C 180,E1 -14160.28,E2 -14160.28} C_VEL
LIN {X 0,Y 340.953,Z 543.1,A -85,B 0,C 180,E1 -14161.365,E2 -14161.365} C_VEL
LIN {X 0,Y 340.743,Z 542.208,A -85,B 0,C 180,E1 -14161.86,E2 -14161.86} C_VEL
LIN {X 0,Y 340.722,Z 542.041,A -85,B 0,C 180,E1 -14165.279,E2 -14165.279} C_VEL
LIN {X 0,Y 340.713,Z 542.043,A -85,B 0,C 180,E1 -14168.387,E2 -14168.387} C_VEL
LIN {X 0,Y 340.703,Z 542.045,A -85,B 0,C 180,E1 -14172.046,E2 -14172.046} C_VEL
LIN {X 0,Y 340.656,Z 542.05,A -85,B 0,C 180,E1 -14176.227,E2 -14176.227} C_VEL
LIN {X 0,Y 340.746,Z 542.217,A -85,B 0,C 180,E1 -14178.607,E2 -14178.607} C_VEL
LIN {X 0,Y 341.338,Z 544.229,A -85,B 0,C 180,E1 -14179.625,E2 -14179.625} C_VEL
LIN {X 0,Y 342.329,Z 545.699,A -85,B 0,C 180,E1 -14180.474,E2 -14180.474} C_VEL
LIN {X 0,Y 345.085,Z 552.234,A -85,B 0,C 180,E1 -14183.18,E2 -14183.18} C_VEL
LIN {X 0,Y 347.569,Z 559.075,A -85,B 0,C 180,E1 -14185.516,E2 -14185.516} C_VEL
LIN {X 0,Y 350.173,Z 568.166,A -85,B 0,C 180,E1 -14188.165,E2 -14188.165} C_VEL
LIN {X 0,Y 351.589,Z 575.463,A -85,B 0,C 180,E1 -14190.018,E2 -14190.018} C_VEL
LIN {X 0,Y 351.765,Z 578.502,A -85,B 0,C 180,E1 -14190.693,E2 -14190.693} C_VEL
LIN {X 0,Y 349.163,Z 599.541,A -85,B 0,C 180,E1 -14194.677,E2 -14194.677} C_VEL
LIN {X 0,Y 346.961,Z 620.579,A -85,B 0,C 180,E1 -14198.617,E2 -14198.617} C_VEL
LIN {X 0,Y 345.971,Z 632.069,A -85,B 0,C 180,E1 -14200.725,E2 -14200.725} C_VEL
LIN {X 0,Y 348.648,Z 647.472,A -85,B 0,C 180,E1 -14201.605,E2 -14201.605} C_VEL
LIN {X 0,Y 349.329,Z 655.763,A -85,B 0,C 180,E1 -14201.975,E2 -14201.975} C_VEL
LIN {X 0,Y 347.034,Z 705.884,A -85,B 0,C 180,E1 -14203.567,E2 -14203.567} C_VEL
LIN {X 0,Y 346.345,Z 716.637,A -85,B 0,C 180,E1 -14204.101,E2 -14204.101} C_VEL
LIN {X 0,Y 345.507,Z 726.85,A -85,B 0,C 180,E1 -14204.818,E2 -14204.818} C_VEL
LIN {X 0,Y 344.565,Z 736.061,A -85,B 0,C 180,E1 -14205.682,E2 -14205.682} C_VEL
LIN {X 0,Y 343.656,Z 744.655,A -85,B 0,C 180,E1 -14206.699,E2 -14206.699} C_VEL
LIN {X 0,Y 342.692,Z 752.507,A -85,B 0,C 180,E1 -14207.865,E2 -14207.865} C_VEL
LIN {X 0,Y 341.838,Z 758.831,A -85,B 0,C 180,E1 -14209.037,E2 -14209.037} C_VEL
LIN {X 0,Y 340.961,Z 765.248,A -85,B 0,C 180,E1 -14210.509,E2 -14210.509} C_VEL
LIN {X 0,Y 340.438,Z 769.342,A -85,B 0,C 180,E1 -14211.691,E2 -14211.691} C_VEL
LIN {X 0,Y 339.99,Z 773.575,A -85,B 0,C 180,E1 -14213.248,E2 -14213.248} C_VEL
LIN {X 0,Y 339.412,Z 777.167,A -85,B 0,C 180,E1 -14215.249,E2 -14215.249} C_VEL
LIN {X 0,Y 339.175,Z 778.501,A -85,B 0,C 180,E1 -14216.436,E2 -14216.436} C_VEL
LIN {X 0,Y 339.046,Z 779.248,A -85,B 0,C 180,E1 -14217.624,E2 -14217.624} C_VEL
LIN {X 0,Y 338.976,Z 779.418,A -85,B 0,C 180,E1 -14218.812,E2 -14218.812} C_VEL
LIN {X 0,Y 338.978,Z 778.994,A -85,B 0,C 180,E1 -14220,E2 -14220} C_VEL
LIN {X 0,Y 338.969,Z 777.954,A -85,B 0,C 180,E1 -14221.188,E2 -14221.188} C_VEL
LIN {X 0,Y 339.065,Z 775.17,A -85,B 0,C 180,E1 -14222.97,E2 -14222.97} C_VEL
LIN {X 0,Y 339.245,Z 770.96,A -85,B 0,C 180,E1 -14224.753,E2 -14224.753} C_VEL
LIN {X 0,Y 339.342,Z 766.238,A -85,B 0,C 180,E1 -14226.215,E2 -14226.215} C_VEL
LIN {X 0,Y 339.707,Z 759.815,A -85,B 0,C 180,E1 -14227.728,E2 -14227.728} C_VEL
LIN {X 0,Y 340.033,Z 753.543,A -85,B 0,C 180,E1 -14228.918,E2 -14228.918} C_VEL
LIN {X 0,Y 340.433,Z 744.725,A -85,B 0,C 180,E1 -14230.257,E2 -14230.257} C_VEL
LIN {X 0,Y 340.973,Z 735.921,A -85,B 0,C 180,E1 -14231.292,E2 -14231.292} C_VEL
LIN {X 0,Y 341.41,Z 726.404,A -85,B 0,C 180,E1 -14232.181,E2 -14232.181} C_VEL
LIN {X 0,Y 341.811,Z 715.597,A -85,B 0,C 180,E1 -14232.921,E2 -14232.921} C_VEL
LIN {X 0,Y 342.162,Z 705.694,A -85,B 0,C 180,E1 -14233.398,E2 -14233.398} C_VEL
LIN {X 0,Y 342.695,Z 680.967,A -85,B 0,C 180,E1 -14234.133,E2 -14234.133} C_VEL
LIN {X 0,Y 343.124,Z 650.323,A -85,B 0,C 180,E1 -14235.002,E2 -14235.002} C_VEL
LIN {X 0,Y 341.549,Z 631.796,A -85,B 0,C 180,E1 -14235.592,E2 -14235.592} C_VEL
LIN {X 0,Y 342.487,Z 613.426,A -85,B 0,C 180,E1 -14238.857,E2 -14238.857} C_VEL
LIN {X 0,Y 343.73,Z 592.833,A -85,B 0,C 180,E1 -14242.543,E2 -14242.543} C_VEL
LIN {X 0,Y 345.211,Z 570.176,A -85,B 0,C 180,E1 -14246.608,E2 -14246.608} C_VEL
LIN {X 0,Y 345.468,Z 564.872,A -85,B 0,C 180,E1 -14247.569,E2 -14247.569} C_VEL
LIN {X 0,Y 342.671,Z 551.016,A -85,B 0,C 180,E1 -14250.261,E2 -14250.261} C_VEL
LIN {X 0,Y 340.776,Z 542.168,A -85,B 0,C 180,E1 -14252.068,E2 -14252.068} C_VEL
LIN {X 0,Y 340.723,Z 542.043,A -85,B 0,C 180,E1 -14255.279,E2 -14255.279} C_VEL
LIN {X 0,Y 340.715,Z 542.047,A -85,B 0,C 180,E1 -14258.386,E2 -14258.386} C_VEL
LIN {X 0,Y 340.703,Z 542.008,A -85,B 0,C 180,E1 -14262.045,E2 -14262.045} C_VEL
LIN {X 0,Y 340.702,Z 542.039,A -85,B 0,C 180,E1 -14265.463,E2 -14265.463} C_VEL
LIN {X 0,Y 340.693,Z 542.034,A -85,B 0,C 180,E1 -14268.69,E2 -14268.69} C_VEL
LIN {X 0,Y 340.737,Z 542.026,A -85,B 0,C 180,E1 -14271.772,E2 -14271.772} C_VEL
LIN {X 0,Y 340.727,Z 542.031,A -85,B 0,C 180,E1 -14275.595,E2 -14275.595} C_VEL
LIN {X 0,Y 340.773,Z 542.038,A -85,B 0,C 180,E1 -14280.02,E2 -14280.02} C_VEL
LIN {X 0,Y 340.848,Z 542.17,A -85,B 0,C 180,E1 -14283.106,E2 -14283.106} C_VEL
LIN {X 0,Y 342.923,Z 552.514,A -85,B 0,C 180,E1 -14286.407,E2 -14286.407} C_VEL
LIN {X 0,Y 343.308,Z 553.925,A -85,B 0,C 180,E1 -14286.557,E2 -14286.557} C_VEL
LIN {X 0,Y 347.609,Z 565.502,A -85,B 0,C 180,E1 -14287.132,E2 -14287.132} C_VEL
LIN {X 0,Y 350.817,Z 581.563,A -85,B 0,C 180,E1 -14287.704,E2 -14287.704} C_VEL
LIN {X 0,Y 349.24,Z 659.086,A -85,B 0,C 180,E1 -14289.302,E2 -14289.302} C_VEL
LIN {X 0,Y 348.636,Z 672.518,A -85,B 0,C 180,E1 -14289.804,E2 -14289.804} C_VEL
LIN {X 0,Y 347.845,Z 685.291,A -85,B 0,C 180,E1 -14290.525,E2 -14290.525} C_VEL
LIN {X 0,Y 346.855,Z 696.621,A -85,B 0,C 180,E1 -14291.389,E2 -14291.389} C_VEL
LIN {X 0,Y 345.73,Z 707.114,A -85,B 0,C 180,E1 -14292.414,E2 -14292.414} C_VEL
LIN {X 0,Y 344.672,Z 717.723,A -85,B 0,C 180,E1 -14293.726,E2 -14293.726} C_VEL
LIN {X 0,Y 343.472,Z 727.266,A -85,B 0,C 180,E1 -14295.18,E2 -14295.18} C_VEL
LIN {X 0,Y 342.372,Z 735.136,A -85,B 0,C 180,E1 -14296.647,E2 -14296.647} C_VEL
LIN {X 0,Y 341.341,Z 742.823,A -85,B 0,C 180,E1 -14298.418,E2 -14298.418} C_VEL
LIN {X 0,Y 340.658,Z 748.071,A -85,B 0,C 180,E1 -14299.899,E2 -14299.899} C_VEL
LIN {X 0,Y 339.994,Z 753.163,A -85,B 0,C 180,E1 -14301.679,E2 -14301.679} C_VEL
LIN {X 0,Y 339.638,Z 756.863,A -85,B 0,C 180,E1 -14303.34,E2 -14303.34} C_VEL
LIN {X 0,Y 339.383,Z 760.023,A -85,B 0,C 180,E1 -14305.248,E2 -14305.248} C_VEL
LIN {X 0,Y 339.192,Z 761.423,A -85,B 0,C 180,E1 -14306.435,E2 -14306.435} C_VEL
LIN {X 0,Y 339.063,Z 763.031,A -85,B 0,C 180,E1 -14308.811,E2 -14308.811} C_VEL
LIN {X 0,Y 339.072,Z 763.263,A -85,B 0,C 180,E1 -14309.999,E2 -14309.999} C_VEL
LIN {X 0,Y 339.062,Z 763.074,A -85,B 0,C 180,E1 -14311.187,E2 -14311.187} C_VEL
LIN {X 0,Y 339.187,Z 761.525,A -85,B 0,C 180,E1 -14313.563,E2 -14313.563} C_VEL
LIN {X 0,Y 339.376,Z 760.168,A -85,B 0,C 180,E1 -14314.75,E2 -14314.75} C_VEL
LIN {X 0,Y 339.634,Z 757.082,A -85,B 0,C 180,E1 -14316.655,E2 -14316.655} C_VEL
LIN {X 0,Y 339.991,Z 753.414,A -85,B 0,C 180,E1 -14318.319,E2 -14318.319} C_VEL
LIN {X 0,Y 340.632,Z 748.4,A -85,B 0,C 180,E1 -14320.099,E2 -14320.099} C_VEL
LIN {X 0,Y 341.435,Z 742.087,A -85,B 0,C 180,E1 -14321.877,E2 -14321.877} C_VEL
LIN {X 0,Y 342.457,Z 734.181,A -85,B 0,C 180,E1 -14323.65,E2 -14323.65} C_VEL
LIN {X 0,Y 343.909,Z 724.341,A -85,B 0,C 180,E1 -14325.405,E2 -14325.405} C_VEL
LIN {X 0,Y 345.033,Z 714.022,A -85,B 0,C 180,E1 -14326.872,E2 -14326.872} C_VEL
LIN {X 0,Y 346.216,Z 702.824,A -85,B 0,C 180,E1 -14328.136,E2 -14328.136} C_VEL
LIN {X 0,Y 347.42,Z 690.754,A -85,B 0,C 180,E1 -14329.19,E2 -14329.19} C_VEL
LIN {X 0,Y 348.4,Z 678.665,A -85,B 0,C 180,E1 -14329.977,E2 -14329.977} C_VEL
LIN {X 0,Y 348.576,Z 674.878,A -85,B 0,C 180,E1 -14330.184,E2 -14330.184} C_VEL
LIN {X 0,Y 348.257,Z 669.249,A -85,B 0,C 180,E1 -14330.483,E2 -14330.483} C_VEL
LIN {X 0,Y 345.959,Z 660.068,A -85,B 0,C 180,E1 -14330.98,E2 -14330.98} C_VEL
LIN {X 0,Y 343.494,Z 650.77,A -85,B 0,C 180,E1 -14331.379,E2 -14331.379} C_VEL
LIN {X 0,Y 343.052,Z 644.963,A -85,B 0,C 180,E1 -14331.535,E2 -14331.535} C_VEL
LIN {X 0,Y 344.175,Z 581.599,A -85,B 0,C 180,E1 -14332.861,E2 -14332.861} C_VEL
LIN {X 0,Y 340.737,Z 565.772,A -85,B 0,C 180,E1 -14333.463,E2 -14333.463} C_VEL
LIN {X 0,Y 335.875,Z 553.116,A -85,B 0,C 180,E1 -14334.161,E2 -14334.161} C_VEL
LIN {X 0,Y 333.874,Z 543.427,A -85,B 0,C 180,E1 -14337.246,E2 -14337.246} C_VEL
LIN {X 0,Y 333.735,Z 542.919,A -85,B 0,C 180,E1 -14337.598,E2 -14337.598} C_VEL
LIN {X 0,Y 333.688,Z 542.907,A -85,B 0,C 180,E1 -14340.362,E2 -14340.362} C_VEL
LIN {X 0,Y 333.672,Z 542.923,A -85,B 0,C 180,E1 -14344.657,E2 -14344.657} C_VEL
LIN {X 0,Y 333.652,Z 542.926,A -85,B 0,C 180,E1 -14347.649,E2 -14347.649} C_VEL
LIN {X 0,Y 333.647,Z 542.917,A -85,B 0,C 180,E1 -14350.766,E2 -14350.766} C_VEL
LIN {X 0,Y 333.59,Z 542.918,A -85,B 0,C 180,E1 -14354.25,E2 -14354.25} C_VEL
LIN {X 0,Y 333.669,Z 542.924,A -85,B 0,C 180,E1 -14357.622,E2 -14357.622} C_VEL
LIN {X 0,Y 333.673,Z 542.898,A -85,B 0,C 180,E1 -14361.195,E2 -14361.195} C_VEL
LIN {X 0,Y 333.687,Z 542.921,A -85,B 0,C 180,E1 -14365.223,E2 -14365.223} C_VEL
LIN {X 0,Y 333.691,Z 542.921,A -85,B 0,C 180,E1 -14369.637,E2 -14369.637} C_VEL
LIN {X 0,Y 333.738,Z 542.901,A -85,B 0,C 180,E1 -14372.4,E2 -14372.4} C_VEL
LIN {X 0,Y 333.72,Z 542.915,A -85,B 0,C 180,E1 -14375.09,E2 -14375.09} C_VEL
LIN {X 0,Y 333.675,Z 542.913,A -85,B 0,C 180,E1 -14379.019,E2 -14379.019} C_VEL
LIN {X 0,Y 333.787,Z 542.905,A -85,B 0,C 180,E1 -14381.589,E2 -14381.589} C_VEL
LIN {X 0,Y 333.801,Z 542.901,A -85,B 0,C 180,E1 -14385.576,E2 -14385.576} C_VEL
LIN {X 0,Y 333.826,Z 542.895,A -85,B 0,C 180,E1 -14389.078,E2 -14389.078} C_VEL
LIN {X 0,Y 334.018,Z 542.875,A -85,B 0,C 180,E1 -14392.747,E2 -14392.747} C_VEL
LIN {X 0,Y 333.806,Z 542.902,A -85,B 0,C 180,E1 -14395.169,E2 -14395.169} C_VEL
LIN {X 0,Y 334.1,Z 542.856,A -85,B 0,C 180,E1 -14397.589,E2 -14397.589} C_VEL
LIN {X 0,Y 334.26,Z 542.848,A -85,B 0,C 180,E1 -14400,E2 -14400} C_VEL
LIN {X 0,Y 334.1,Z 542.859,A -85,B 0,C 180,E1 -14402.411,E2 -14402.411} C_VEL
LIN {X 0,Y 334.016,Z 542.878,A -85,B 0,C 180,E1 -14406.039,E2 -14406.039} C_VEL
LIN {X 0,Y 333.977,Z 542.877,A -85,B 0,C 180,E1 -14408.501,E2 -14408.501} C_VEL
LIN {X 0,Y 333.788,Z 542.905,A -85,B 0,C 180,E1 -14412.155,E2 -14412.155} C_VEL
LIN {X 0,Y 333.77,Z 542.898,A -85,B 0,C 180,E1 -14415.887,E2 -14415.887} C_VEL
LIN {X 0,Y 333.79,Z 542.904,A -85,B 0,C 180,E1 -14418.656,E2 -14418.656} C_VEL
LIN {X 0,Y 333.685,Z 542.914,A -85,B 0,C 180,E1 -14422.279,E2 -14422.279} C_VEL
LIN {X 0,Y 333.728,Z 542.905,A -85,B 0,C 180,E1 -14426.247,E2 -14426.247} C_VEL
LIN {X 0,Y 333.683,Z 542.919,A -85,B 0,C 180,E1 -14428.975,E2 -14428.975} C_VEL
LIN {X 0,Y 333.639,Z 542.924,A -85,B 0,C 180,E1 -14432.588,E2 -14432.588} C_VEL
LIN {X 0,Y 333.67,Z 542.899,A -85,B 0,C 180,E1 -14436.14,E2 -14436.14} C_VEL
LIN {X 0,Y 333.642,Z 542.923,A -85,B 0,C 180,E1 -14439.193,E2 -14439.193} C_VEL
LIN {X 0,Y 333.636,Z 542.91,A -85,B 0,C 180,E1 -14442.503,E2 -14442.503} C_VEL
LIN {X 0,Y 333.668,Z 542.916,A -85,B 0,C 180,E1 -14445.969,E2 -14445.969} C_VEL
LIN {X 0,Y 333.697,Z 542.92,A -85,B 0,C 180,E1 -14449.306,E2 -14449.306} C_VEL
LIN {X 0,Y 333.662,Z 542.899,A -85,B 0,C 180,E1 -14453.169,E2 -14453.169} C_VEL
LIN {X 0,Y 333.671,Z 542.919,A -85,B 0,C 180,E1 -14455.343,E2 -14455.343} C_VEL
LIN {X 0,Y 333.71,Z 543.01,A -85,B 0,C 180,E1 -14458.317,E2 -14458.317} C_VEL
LIN {X 0,Y 336.044,Z 553.399,A -85,B 0,C 180,E1 -14461.449,E2 -14461.449} C_VEL
LIN {X 0,Y 337.849,Z 562.707,A -85,B 0,C 180,E1 -14464.099,E2 -14464.099} C_VEL
LIN {X 0,Y 338.032,Z 566.442,A -85,B 0,C 180,E1 -14465.103,E2 -14465.103} C_VEL
LIN {X 0,Y 337.585,Z 570.176,A -85,B 0,C 180,E1 -14465.997,E2 -14465.997} C_VEL
LIN {X 0,Y 339.366,Z 579.979,A -85,B 0,C 180,E1 -14466.396,E2 -14466.396} C_VEL
LIN {X 0,Y 343.744,Z 606.888,A -85,B 0,C 180,E1 -14467.309,E2 -14467.309} C_VEL
LIN {X 0,Y 342.428,Z 678.458,A -85,B 0,C 180,E1 -14468.834,E2 -14468.834} C_VEL
LIN {X 0,Y 341.573,Z 691.637,A -85,B 0,C 180,E1 -14469.331,E2 -14469.331} C_VEL
LIN {X 0,Y 340.688,Z 703.761,A -85,B 0,C 180,E1 -14470.023,E2 -14470.023} C_VEL
LIN {X 0,Y 339.466,Z 716.005,A -85,B 0,C 180,E1 -14470.971,E2 -14470.971} C_VEL
LIN {X 0,Y 338.107,Z 727.584,A -85,B 0,C 180,E1 -14472.147,E2 -14472.147} C_VEL
LIN {X 0,Y 336.762,Z 738.29,A -85,B 0,C 180,E1 -14473.522,E2 -14473.522} C_VEL
LIN {X 0,Y 335.739,Z 746.546,A -85,B 0,C 180,E1 -14474.833,E2 -14474.833} C_VEL
LIN {X 0,Y 334.705,Z 754.418,A -85,B 0,C 180,E1 -14476.338,E2 -14476.338} C_VEL
LIN {X 0,Y 333.601,Z 762.106,A -85,B 0,C 180,E1 -14478.148,E2 -14478.148} C_VEL
LIN {X 0,Y 333.006,Z 767.379,A -85,B 0,C 180,E1 -14479.667,E2 -14479.667} C_VEL
LIN {X 0,Y 332.478,Z 772.489,A -85,B 0,C 180,E1 -14481.492,E2 -14481.492} C_VEL
LIN {X 0,Y 332.107,Z 776.461,A -85,B 0,C 180,E1 -14483.317,E2 -14483.317} C_VEL
LIN {X 0,Y 331.981,Z 779.399,A -85,B 0,C 180,E1 -14485.144,E2 -14485.144} C_VEL
LIN {X 0,Y 331.996,Z 780.797,A -85,B 0,C 180,E1 -14486.36,E2 -14486.36} C_VEL
LIN {X 0,Y 331.929,Z 783.862,A -85,B 0,C 180,E1 -14490.001,E2 -14490.001} C_VEL
LIN {X 0,Y 331.883,Z 784.379,A -85,B 0,C 180,E1 -14491.214,E2 -14491.214} C_VEL
LIN {X 0,Y 331.915,Z 784.304,A -85,B 0,C 180,E1 -14492.428,E2 -14492.428} C_VEL
LIN {X 0,Y 332.013,Z 783.636,A -85,B 0,C 180,E1 -14493.642,E2 -14493.642} C_VEL
LIN {X 0,Y 332.097,Z 782.372,A -85,B 0,C 180,E1 -14494.857,E2 -14494.857} C_VEL
LIN {X 0,Y 332.241,Z 779.275,A -85,B 0,C 180,E1 -14496.682,E2 -14496.682} C_VEL
LIN {X 0,Y 332.616,Z 774.738,A -85,B 0,C 180,E1 -14498.507,E2 -14498.507} C_VEL
LIN {X 0,Y 332.984,Z 769.58,A -85,B 0,C 180,E1 -14500.029,E2 -14500.029} C_VEL
LIN {X 0,Y 334.485,Z 755.719,A -85,B 0,C 180,E1 -14503.364,E2 -14503.364} C_VEL
LIN {X 0,Y 335.485,Z 748.128,A -85,B 0,C 180,E1 -14504.871,E2 -14504.871} C_VEL
LIN {X 0,Y 336.733,Z 738.212,A -85,B 0,C 180,E1 -14506.475,E2 -14506.475} C_VEL
LIN {X 0,Y 338.076,Z 727.433,A -85,B 0,C 180,E1 -14507.857,E2 -14507.857} C_VEL
LIN {X 0,Y 339.478,Z 715.82,A -85,B 0,C 180,E1 -14509.031,E2 -14509.031} C_VEL
LIN {X 0,Y 340.673,Z 703.504,A -85,B 0,C 180,E1 -14509.98,E2 -14509.98} C_VEL
LIN {X 0,Y 341.689,Z 690.528,A -85,B 0,C 180,E1 -14510.704,E2 -14510.704} C_VEL
LIN {X 0,Y 342.379,Z 677.909,A -85,B 0,C 180,E1 -14511.172,E2 -14511.172} C_VEL
LIN {X 0,Y 343.739,Z 607.093,A -85,B 0,C 180,E1 -14512.67,E2 -14512.67} C_VEL
LIN {X 0,Y 341.855,Z 594.056,A -85,B 0,C 180,E1 -14513.127,E2 -14513.127} C_VEL
LIN {X 0,Y 342.517,Z 581.806,A -85,B 0,C 180,E1 -14514.405,E2 -14514.405} C_VEL
LIN {X 0,Y 342.095,Z 575.146,A -85,B 0,C 180,E1 -14515.319,E2 -14515.319} C_VEL
LIN {X 0,Y 341.546,Z 568.931,A -85,B 0,C 180,E1 -14516.295,E2 -14516.295} C_VEL
LIN {X 0,Y 338.744,Z 557.715,A -85,B 0,C 180,E1 -14518.842,E2 -14518.842} C_VEL
LIN {X 0,Y 337.262,Z 550.81,A -85,B 0,C 180,E1 -14520.782,E2 -14520.782} C_VEL
LIN {X 0,Y 336.781,Z 548.908,A -85,B 0,C 180,E1 -14521.448,E2 -14521.448} C_VEL
LIN {X 0,Y 335.935,Z 547.354,A -85,B 0,C 180,E1 -14522.231,E2 -14522.231} C_VEL
LIN {X 0,Y 334.249,Z 544.981,A -85,B 0,C 180,E1 -14523.863,E2 -14523.863} C_VEL
LIN {X 0,Y 333.719,Z 543.075,A -85,B 0,C 180,E1 -14525.302,E2 -14525.302} C_VEL
LIN {X 0,Y 333.651,Z 542.922,A -85,B 0,C 180,E1 -14529.193,E2 -14529.193} C_VEL
LIN {X 0,Y 333.636,Z 542.923,A -85,B 0,C 180,E1 -14532.5,E2 -14532.5} C_VEL
LIN {X 0,Y 333.666,Z 543.258,A -85,B 0,C 180,E1 -14535.467,E2 -14535.467} C_VEL
LIN {X 0,Y 335.059,Z 546.354,A -85,B 0,C 180,E1 -14537.839,E2 -14537.839} C_VEL
LIN {X 0,Y 337.329,Z 550.837,A -85,B 0,C 180,E1 -14540.433,E2 -14540.433} C_VEL
LIN {X 0,Y 339.141,Z 555.254,A -85,B 0,C 180,E1 -14542.399,E2 -14542.399} C_VEL
LIN {X 0,Y 341.486,Z 561.738,A -85,B 0,C 180,E1 -14544.812,E2 -14544.812} C_VEL
LIN {X 0,Y 343.734,Z 569.526,A -85,B 0,C 180,E1 -14547.254,E2 -14547.254} C_VEL
LIN {X 0,Y 345.375,Z 577.539,A -85,B 0,C 180,E1 -14549.421,E2 -14549.421} C_VEL
LIN {X 0,Y 345.648,Z 580.396,A -85,B 0,C 180,E1 -14550.122,E2 -14550.122} C_VEL
LIN {X 0,Y 344.196,Z 591.652,A -85,B 0,C 180,E1 -14552.321,E2 -14552.321} C_VEL
LIN {X 0,Y 341.6,Z 612.6,A -85,B 0,C 180,E1 -14556.347,E2 -14556.347} C_VEL
LIN {X 0,Y 339.608,Z 632.354,A -85,B 0,C 180,E1 -14560.054,E2 -14560.054} C_VEL
LIN {X 0,Y 342.45,Z 648.106,A -85,B 0,C 180,E1 -14561.011,E2 -14561.011} C_VEL
LIN {X 0,Y 343.184,Z 656.083,A -85,B 0,C 180,E1 -14561.393,E2 -14561.393} C_VEL
LIN {X 0,Y 340.735,Z 705.808,A -85,B 0,C 180,E1 -14563.023,E2 -14563.023} C_VEL
LIN {X 0,Y 339.977,Z 716.446,A -85,B 0,C 180,E1 -14563.564,E2 -14563.564} C_VEL
LIN {X 0,Y 338.987,Z 727.463,A -85,B 0,C 180,E1 -14564.364,E2 -14564.364} C_VEL
LIN {X 0,Y 337.98,Z 736.567,A -85,B 0,C 180,E1 -14565.243,E2 -14565.243} C_VEL
LIN {X 0,Y 336.874,Z 746.196,A -85,B 0,C 180,E1 -14566.426,E2 -14566.426} C_VEL
LIN {X 0,Y 335.834,Z 753.691,A -85,B 0,C 180,E1 -14567.614,E2 -14567.614} C_VEL
LIN {X 0,Y 334.938,Z 759.838,A -85,B 0,C 180,E1 -14568.808,E2 -14568.808} C_VEL
LIN {X 0,Y 334.022,Z 766.068,A -85,B 0,C 180,E1 -14570.31,E2 -14570.31} C_VEL
LIN {X 0,Y 333.467,Z 770.004,A -85,B 0,C 180,E1 -14571.516,E2 -14571.516} C_VEL
LIN {X 0,Y 332.935,Z 774.198,A -85,B 0,C 180,E1 -14573.185,E2 -14573.185} C_VEL
LIN {X 0,Y 332.754,Z 775.655,A -85,B 0,C 180,E1 -14573.938,E2 -14573.938} C_VEL
LIN {X 0,Y 332.367,Z 777.496,A -85,B 0,C 180,E1 -14575.148,E2 -14575.148} C_VEL
LIN {X 0,Y 332.109,Z 778.724,A -85,B 0,C 180,E1 -14576.36,E2 -14576.36} C_VEL
LIN {X 0,Y 331.964,Z 779.364,A -85,B 0,C 180,E1 -14577.573,E2 -14577.573} C_VEL
LIN {X 0,Y 331.886,Z 779.423,A -85,B 0,C 180,E1 -14578.787,E2 -14578.787} C_VEL
LIN {X 0,Y 331.884,Z 778.899,A -85,B 0,C 180,E1 -14580,E2 -14580} C_VEL
LIN {X 0,Y 331.878,Z 777.783,A -85,B 0,C 180,E1 -14581.213,E2 -14581.213} C_VEL
LIN {X 0,Y 331.937,Z 776.045,A -85,B 0,C 180,E1 -14582.427,E2 -14582.427} C_VEL
LIN {X 0,Y 332.082,Z 773.645,A -85,B 0,C 180,E1 -14583.64,E2 -14583.64} C_VEL
LIN {X 0,Y 332.148,Z 769.251,A -85,B 0,C 180,E1 -14585.263,E2 -14585.263} C_VEL
LIN {X 0,Y 332.343,Z 764.503,A -85,B 0,C 180,E1 -14586.618,E2 -14586.618} C_VEL
LIN {X 0,Y 332.642,Z 758.963,A -85,B 0,C 180,E1 -14587.894,E2 -14587.894} C_VEL
LIN {X 0,Y 333.088,Z 750.659,A -85,B 0,C 180,E1 -14589.411,E2 -14589.411} C_VEL
LIN {X 0,Y 333.547,Z 742.085,A -85,B 0,C 180,E1 -14590.624,E2 -14590.624} C_VEL
LIN {X 0,Y 334.112,Z 732.725,A -85,B 0,C 180,E1 -14591.681,E2 -14591.681} C_VEL
LIN {X 0,Y 334.525,Z 722.932,A -85,B 0,C 180,E1 -14592.513,E2 -14592.513} C_VEL
LIN {X 0,Y 334.821,Z 713.552,A -85,B 0,C 180,E1 -14593.118,E2 -14593.118} C_VEL
LIN {X 0,Y 335.169,Z 701.675,A -85,B 0,C 180,E1 -14593.645,E2 -14593.645} C_VEL
LIN {X 0,Y 336.097,Z 651.039,A -85,B 0,C 180,E1 -14595.126,E2 -14595.126} C_VEL
LIN {X 0,Y 334.517,Z 632.009,A -85,B 0,C 180,E1 -14595.754,E2 -14595.754} C_VEL
LIN {X 0,Y 335.417,Z 615.841,A -85,B 0,C 180,E1 -14598.635,E2 -14598.635} C_VEL
LIN {X 0,Y 336.749,Z 593.393,A -85,B 0,C 180,E1 -14602.712,E2 -14602.712} C_VEL
LIN {X 0,Y 338.409,Z 568.8,A -85,B 0,C 180,E1 -14607.187,E2 -14607.187} C_VEL
LIN {X 0,Y 338.367,Z 565.166,A -85,B 0,C 180,E1 -14607.862,E2 -14607.862} C_VEL
LIN {X 0,Y 334.979,Z 548.684,A -85,B 0,C 180,E1 -14611.123,E2 -14611.123} C_VEL
LIN {X 0,Y 333.718,Z 543.055,A -85,B 0,C 180,E1 -14612.303,E2 -14612.303} C_VEL
LIN {X 0,Y 333.681,Z 542.922,A -85,B 0,C 180,E1 -14616.139,E2 -14616.139} C_VEL
LIN {X 0,Y 333.652,Z 542.919,A -85,B 0,C 180,E1 -14619.192,E2 -14619.192} C_VEL
LIN {X 0,Y 333.637,Z 542.884,A -85,B 0,C 180,E1 -14622.5,E2 -14622.5} C_VEL
LIN {X 0,Y 333.651,Z 542.919,A -85,B 0,C 180,E1 -14625.963,E2 -14625.963} C_VEL
LIN {X 0,Y 333.652,Z 542.904,A -85,B 0,C 180,E1 -14629.315,E2 -14629.315} C_VEL
LIN {X 0,Y 333.669,Z 542.922,A -85,B 0,C 180,E1 -14633.167,E2 -14633.167} C_VEL
LIN {X 0,Y 333.678,Z 542.909,A -85,B 0,C 180,E1 -14635.341,E2 -14635.341} C_VEL
LIN {X 0,Y 333.709,Z 542.916,A -85,B 0,C 180,E1 -14639.709,E2 -14639.709} C_VEL
LIN {X 0,Y 333.794,Z 543.136,A -85,B 0,C 180,E1 -14642.744,E2 -14642.744} C_VEL
LIN {X 0,Y 335.814,Z 552.823,A -85,B 0,C 180,E1 -14645.894,E2 -14645.894} C_VEL
LIN {X 0,Y 336.353,Z 554.575,A -85,B 0,C 180,E1 -14646.058,E2 -14646.058} C_VEL
LIN {X 0,Y 341.278,Z 567.586,A -85,B 0,C 180,E1 -14646.725,E2 -14646.725} C_VEL
LIN {X 0,Y 344.254,Z 582.997,A -85,B 0,C 180,E1 -14647.283,E2 -14647.283} C_VEL
LIN {X 0,Y 342.628,Z 659.308,A -85,B 0,C 180,E1 -14648.884,E2 -14648.884} C_VEL
LIN {X 0,Y 342.006,Z 672.733,A -85,B 0,C 180,E1 -14649.395,E2 -14649.395} C_VEL
LIN {X 0,Y 341.17,Z 685.503,A -85,B 0,C 180,E1 -14650.129,E2 -14650.129} C_VEL
LIN {X 0,Y 340.148,Z 696.831,A -85,B 0,C 180,E1 -14651.008,E2 -14651.008} C_VEL
LIN {X 0,Y 338.979,Z 707.323,A -85,B 0,C 180,E1 -14652.052,E2 -14652.052} C_VEL
LIN {X 0,Y 337.928,Z 717.116,A -85,B 0,C 180,E1 -14653.273,E2 -14653.273} C_VEL
LIN {X 0,Y 336.618,Z 727.474,A -85,B 0,C 180,E1 -14654.871,E2 -14654.871} C_VEL
LIN {X 0,Y 335.473,Z 735.344,A -85,B 0,C 180,E1 -14656.367,E2 -14656.367} C_VEL
LIN {X 0,Y 334.389,Z 743.03,A -85,B 0,C 180,E1 -14658.174,E2 -14658.174} C_VEL
LIN {X 0,Y 333.666,Z 748.278,A -85,B 0,C 180,E1 -14659.685,E2 -14659.685} C_VEL
LIN {X 0,Y 332.949,Z 753.369,A -85,B 0,C 180,E1 -14661.502,E2 -14661.502} C_VEL
LIN {X 0,Y 332.553,Z 757.368,A -85,B 0,C 180,E1 -14663.353,E2 -14663.353} C_VEL
LIN {X 0,Y 332.304,Z 760.228,A -85,B 0,C 180,E1 -14665.146,E2 -14665.146} C_VEL
LIN {X 0,Y 332.123,Z 761.627,A -85,B 0,C 180,E1 -14666.359,E2 -14666.359} C_VEL
LIN {X 0,Y 331.968,Z 763.235,A -85,B 0,C 180,E1 -14668.786,E2 -14668.786} C_VEL
LIN {X 0,Y 331.975,Z 763.467,A -85,B 0,C 180,E1 -14669.999,E2 -14669.999} C_VEL
LIN {X 0,Y 331.968,Z 763.278,A -85,B 0,C 180,E1 -14671.212,E2 -14671.212} C_VEL
LIN {X 0,Y 332.118,Z 761.729,A -85,B 0,C 180,E1 -14673.639,E2 -14673.639} C_VEL
LIN {X 0,Y 332.298,Z 760.372,A -85,B 0,C 180,E1 -14674.852,E2 -14674.852} C_VEL
LIN {X 0,Y 332.548,Z 757.564,A -85,B 0,C 180,E1 -14676.64,E2 -14676.64} C_VEL
LIN {X 0,Y 332.944,Z 753.618,A -85,B 0,C 180,E1 -14678.496,E2 -14678.496} C_VEL
LIN {X 0,Y 333.642,Z 748.603,A -85,B 0,C 180,E1 -14680.313,E2 -14680.313} C_VEL
LIN {X 0,Y 334.495,Z 742.289,A -85,B 0,C 180,E1 -14682.127,E2 -14682.127} C_VEL
LIN {X 0,Y 335.553,Z 734.383,A -85,B 0,C 180,E1 -14683.936,E2 -14683.936} C_VEL
LIN {X 0,Y 337.083,Z 724.542,A -85,B 0,C 180,E1 -14685.725,E2 -14685.725} C_VEL
LIN {X 0,Y 338.262,Z 714.222,A -85,B 0,C 180,E1 -14687.22,E2 -14687.22} C_VEL
LIN {X 0,Y 339.363,Z 703.993,A -85,B 0,C 180,E1 -14688.409,E2 -14688.409} C_VEL
LIN {X 0,Y 340.552,Z 692.79,A -85,B 0,C 180,E1 -14689.436,E2 -14689.436} C_VEL
LIN {X 0,Y 341.632,Z 680.159,A -85,B 0,C 180,E1 -14690.312,E2 -14690.312} C_VEL
LIN {X 0,Y 342.328,Z 667.509,A -85,B 0,C 180,E1 -14690.936,E2 -14690.936} C_VEL
LIN {X 0,Y 342.88,Z 654.496,A -85,B 0,C 180,E1 -14691.334,E2 -14691.334} C_VEL
LIN {X 0,Y 343.052,Z 644.963,A -85,B 0,C 180,E1 -14691.535,E2 -14691.535} C_VEL
LIN {X 0,Y 342.646,Z 639.152,A -85,B 0,C 180,E1 -14691.691,E2 -14691.691} C_VEL
LIN {X 0,Y 337.696,Z 620.464,A -85,B 0,C 180,E1 -14692.449,E2 -14692.449} C_VEL
LIN {X 0,Y 337.114,Z 614.656,A -85,B 0,C 180,E1 -14692.622,E2 -14692.622} C_VEL
LIN {X 0,Y 337.606,Z 582.596,A -85,B 0,C 180,E1 -14693.313,E2 -14693.313} C_VEL
LIN {X 0,Y 334.508,Z 568.133,A -85,B 0,C 180,E1 -14693.877,E2 -14693.877} C_VEL
LIN {X 0,Y 328.731,Z 553.534,A -85,B 0,C 180,E1 -14694.703,E2 -14694.703} C_VEL
LIN {X 0,Y 328.447,Z 552.211,A -85,B 0,C 180,E1 -14695.009,E2 -14695.009} C_VEL
LIN {X 0,Y 326.704,Z 543.961,A -85,B 0,C 180,E1 -14697.821,E2 -14697.821} C_VEL
LIN {X 0,Y 326.589,Z 543.801,A -85,B 0,C 180,E1 -14701.094,E2 -14701.094} C_VEL
LIN {X 0,Y 326.605,Z 543.804,A -85,B 0,C 180,E1 -14704.018,E2 -14704.018} C_VEL
LIN {X 0,Y 326.627,Z 543.797,A -85,B 0,C 180,E1 -14707.238,E2 -14707.238} C_VEL
LIN {X 0,Y 326.578,Z 543.8,A -85,B 0,C 180,E1 -14711.131,E2 -14711.131} C_VEL
LIN {X 0,Y 326.526,Z 543.795,A -85,B 0,C 180,E1 -14714.742,E2 -14714.742} C_VEL
LIN {X 0,Y 326.593,Z 543.802,A -85,B 0,C 180,E1 -14718.157,E2 -14718.157} C_VEL
LIN {X 0,Y 326.639,Z 543.773,A -85,B 0,C 180,E1 -14721.393,E2 -14721.393} C_VEL
LIN {X 0,Y 326.62,Z 543.799,A -85,B 0,C 180,E1 -14724.849,E2 -14724.849} C_VEL
LIN {X 0,Y 326.605,Z 543.796,A -85,B 0,C 180,E1 -14727.455,E2 -14727.455} C_VEL
LIN {X 0,Y 326.655,Z 543.794,A -85,B 0,C 180,E1 -14730.34,E2 -14730.34} C_VEL
LIN {X 0,Y 326.683,Z 543.789,A -85,B 0,C 180,E1 -14734.516,E2 -14734.516} C_VEL
LIN {X 0,Y 326.64,Z 543.787,A -85,B 0,C 180,E1 -14738.545,E2 -14738.545} C_VEL
LIN {X 0,Y 326.737,Z 543.785,A -85,B 0,C 180,E1 -14741.177,E2 -14741.177} C_VEL
LIN {X 0,Y 326.756,Z 543.777,A -85,B 0,C 180,E1 -14745.433,E2 -14745.433} C_VEL
LIN {X 0,Y 326.762,Z 543.776,A -85,B 0,C 180,E1 -14748.839,E2 -14748.839} C_VEL
LIN {X 0,Y 326.972,Z 543.753,A -85,B 0,C 180,E1 -14752.59,E2 -14752.59} C_VEL
LIN {X 0,Y 326.773,Z 543.779,A -85,B 0,C 180,E1 -14755.065,E2 -14755.065} C_VEL
LIN {X 0,Y 327.041,Z 543.735,A -85,B 0,C 180,E1 -14757.537,E2 -14757.537} C_VEL
LIN {X 0,Y 327.211,Z 543.726,A -85,B 0,C 180,E1 -14760,E2 -14760} C_VEL
LIN {X 0,Y 327.041,Z 543.738,A -85,B 0,C 180,E1 -14762.463,E2 -14762.463} C_VEL
LIN {X 0,Y 326.991,Z 543.752,A -85,B 0,C 180,E1 -14766.169,E2 -14766.169} C_VEL
LIN {X 0,Y 326.907,Z 543.758,A -85,B 0,C 180,E1 -14768.655,E2 -14768.655} C_VEL
LIN {X 0,Y 326.73,Z 543.783,A -85,B 0,C 180,E1 -14772.421,E2 -14772.421} C_VEL
LIN {X 0,Y 326.747,Z 543.78,A -85,B 0,C 180,E1 -14774.958,E2 -14774.958} C_VEL
LIN {X 0,Y 326.728,Z 543.784,A -85,B 0,C 180,E1 -14778.84,E2 -14778.84} C_VEL
LIN {X 0,Y 326.614,Z 543.794,A -85,B 0,C 180,E1 -14782.788,E2 -14782.788} C_VEL
LIN {X 0,Y 326.683,Z 543.79,A -85,B 0,C 180,E1 -14785.484,E2 -14785.484} C_VEL
LIN {X 0,Y 326.641,Z 543.797,A -85,B 0,C 180,E1 -14789.661,E2 -14789.661} C_VEL
LIN {X 0,Y 326.613,Z 543.8,A -85,B 0,C 180,E1 -14792.947,E2 -14792.947} C_VEL
LIN {X 0,Y 326.606,Z 543.784,A -85,B 0,C 180,E1 -14795.521,E2 -14795.521} C_VEL
LIN {X 0,Y 326.606,Z 543.8,A -85,B 0,C 180,E1 -14799.228,E2 -14799.228} C_VEL
LIN {X 0,Y 326.587,Z 543.789,A -85,B 0,C 180,E1 -14802.976,E2 -14802.976} C_VEL
LIN {X 0,Y 326.623,Z 543.789,A -85,B 0,C 180,E1 -14807.019,E2 -14807.019} C_VEL
LIN {X 0,Y 326.641,Z 543.779,A -85,B 0,C 180,E1 -14810.767,E2 -14810.767} C_VEL
LIN {X 0,Y 326.61,Z 543.801,A -85,B 0,C 180,E1 -14814.482,E2 -14814.482} C_VEL
LIN {X 0,Y 326.622,Z 543.838,A -85,B 0,C 180,E1 -14817.824,E2 -14817.824} C_VEL
LIN {X 0,Y 328.912,Z 553.821,A -85,B 0,C 180,E1 -14820.947,E2 -14820.947} C_VEL
LIN {X 0,Y 330.852,Z 563.743,A -85,B 0,C 180,E1 -14823.848,E2 -14823.848} C_VEL
LIN {X 0,Y 331.149,Z 567.479,A -85,B 0,C 180,E1 -14824.885,E2 -14824.885} C_VEL
LIN {X 0,Y 330.842,Z 570.108,A -85,B 0,C 180,E1 -14825.491,E2 -14825.491} C_VEL
LIN {X 0,Y 335.506,Z 596.549,A -85,B 0,C 180,E1 -14826.489,E2 -14826.489} C_VEL
LIN {X 0,Y 337.258,Z 609.014,A -85,B 0,C 180,E1 -14826.9,E2 -14826.9} C_VEL
LIN {X 0,Y 335.823,Z 678.266,A -85,B 0,C 180,E1 -14828.397,E2 -14828.397} C_VEL
LIN {X 0,Y 334.945,Z 691.441,A -85,B 0,C 180,E1 -14828.902,E2 -14828.902} C_VEL
LIN {X 0,Y 334.012,Z 703.562,A -85,B 0,C 180,E1 -14829.606,E2 -14829.606} C_VEL
LIN {X 0,Y 332.754,Z 715.805,A -85,B 0,C 180,E1 -14830.572,E2 -14830.572} C_VEL
LIN {X 0,Y 331.355,Z 727.383,A -85,B 0,C 180,E1 -14831.77,E2 -14831.77} C_VEL
LIN {X 0,Y 329.948,Z 737.813,A -85,B 0,C 180,E1 -14833.131,E2 -14833.131} C_VEL
LIN {X 0,Y 328.882,Z 746.343,A -85,B 0,C 180,E1 -14834.508,E2 -14834.508} C_VEL
LIN {X 0,Y 327.799,Z 754.215,A -85,B 0,C 180,E1 -14836.044,E2 -14836.044} C_VEL
LIN {X 0,Y 326.631,Z 761.902,A -85,B 0,C 180,E1 -14837.891,E2 -14837.891} C_VEL
LIN {X 0,Y 325.785,Z 768.997,A -85,B 0,C 180,E1 -14840.063,E2 -14840.063} C_VEL
LIN {X 0,Y 325.287,Z 773.719,A -85,B 0,C 180,E1 -14841.928,E2 -14841.928} C_VEL
LIN {X 0,Y 324.96,Z 777.331,A -85,B 0,C 180,E1 -14843.793,E2 -14843.793} C_VEL
LIN {X 0,Y 324.89,Z 779.195,A -85,B 0,C 180,E1 -14845.037,E2 -14845.037} C_VEL
LIN {X 0,Y 324.9,Z 780.592,A -85,B 0,C 180,E1 -14846.28,E2 -14846.28} C_VEL
LIN {X 0,Y 324.819,Z 782.437,A -85,B 0,C 180,E1 -14848.761,E2 -14848.761} C_VEL
LIN {X 0,Y 324.835,Z 783.631,A -85,B 0,C 180,E1 -14850.001,E2 -14850.001} C_VEL
LIN {X 0,Y 324.794,Z 784.262,A -85,B 0,C 180,E1 -14851.241,E2 -14851.241} C_VEL
LIN {X 0,Y 324.836,Z 784.298,A -85,B 0,C 180,E1 -14852.481,E2 -14852.481} C_VEL
LIN {X 0,Y 324.945,Z 783.74,A -85,B 0,C 180,E1 -14853.721,E2 -14853.721} C_VEL
LIN {X 0,Y 325.024,Z 782.597,A -85,B 0,C 180,E1 -14854.963,E2 -14854.963} C_VEL
LIN {X 0,Y 325.112,Z 780.836,A -85,B 0,C 180,E1 -14856.206,E2 -14856.206} C_VEL
LIN {X 0,Y 325.46,Z 776.888,A -85,B 0,C 180,E1 -14858.07,E2 -14858.07} C_VEL
LIN {X 0,Y 325.798,Z 773.4,A -85,B 0,C 180,E1 -14859.312,E2 -14859.312} C_VEL
LIN {X 0,Y 326.239,Z 767.899,A -85,B 0,C 180,E1 -14860.866,E2 -14860.866} C_VEL
LIN {X 0,Y 326.874,Z 760.177,A -85,B 0,C 180,E1 -14862.575,E2 -14862.575} C_VEL
LIN {X 0,Y 328.171,Z 751.145,A -85,B 0,C 180,E1 -14864.575,E2 -14864.575} C_VEL
LIN {X 0,Y 329.393,Z 741.857,A -85,B 0,C 180,E1 -14866.233,E2 -14866.233} C_VEL
LIN {X 0,Y 330.65,Z 732.144,A -85,B 0,C 180,E1 -14867.632,E2 -14867.632} C_VEL
LIN {X 0,Y 332.164,Z 720.325,A -85,B 0,C 180,E1 -14868.985,E2 -14868.985} C_VEL
LIN {X 0,Y 333.517,Z 708.439,A -85,B 0,C 180,E1 -14870.026,E2 -14870.026} C_VEL
LIN {X 0,Y 334.604,Z 696.066,A -85,B 0,C 180,E1 -14870.841,E2 -14870.841} C_VEL
LIN {X 0,Y 335.533,Z 683.33,A -85,B 0,C 180,E1 -14871.423,E2 -14871.423} C_VEL
LIN {X 0,Y 335.984,Z 669.9,A -85,B 0,C 180,E1 -14871.796,E2 -14871.796} C_VEL
LIN {X 0,Y 337.177,Z 607.872,A -85,B 0,C 180,E1 -14873.114,E2 -14873.114} C_VEL
LIN {X 0,Y 336.074,Z 599.927,A -85,B 0,C 180,E1 -14873.412,E2 -14873.412} C_VEL
LIN {X 0,Y 337.152,Z 585.163,A -85,B 0,C 180,E1 -14874.969,E2 -14874.969} C_VEL
LIN {X 0,Y 336.863,Z 578.022,A -85,B 0,C 180,E1 -14875.985,E2 -14875.985} C_VEL
LIN {X 0,Y 336.654,Z 573.451,A -85,B 0,C 180,E1 -14876.707,E2 -14876.707} C_VEL
LIN {X 0,Y 334.267,Z 563.083,A -85,B 0,C 180,E1 -14879.108,E2 -14879.108} C_VEL
LIN {X 0,Y 332.922,Z 556.295,A -85,B 0,C 180,E1 -14881.032,E2 -14881.032} C_VEL
LIN {X 0,Y 332.218,Z 553.912,A -85,B 0,C 180,E1 -14881.93,E2 -14881.93} C_VEL
LIN {X 0,Y 330.178,Z 550.835,A -85,B 0,C 180,E1 -14883.887,E2 -14883.887} C_VEL
LIN {X 0,Y 329.478,Z 548.892,A -85,B 0,C 180,E1 -14885.166,E2 -14885.166} C_VEL
LIN {X 0,Y 328.032,Z 547.247,A -85,B 0,C 180,E1 -14887.56,E2 -14887.56} C_VEL
LIN {X 0,Y 327.484,Z 546.486,A -85,B 0,C 180,E1 -14890.078,E2 -14890.078} C_VEL
LIN {X 0,Y 327.573,Z 546.635,A -85,B 0,C 180,E1 -14891.691,E2 -14891.691} C_VEL
LIN {X 0,Y 328.921,Z 548.399,A -85,B 0,C 180,E1 -14895.162,E2 -14895.162} C_VEL
LIN {X 0,Y 331.085,Z 553.279,A -85,B 0,C 180,E1 -14898.849,E2 -14898.849} C_VEL
LIN {X 0,Y 333.364,Z 558.57,A -85,B 0,C 180,E1 -14901.609,E2 -14901.609} C_VEL
LIN {X 0,Y 335.591,Z 564.658,A -85,B 0,C 180,E1 -14904.099,E2 -14904.099} C_VEL
LIN {X 0,Y 337.749,Z 572.503,A -85,B 0,C 180,E1 -14906.715,E2 -14906.715} C_VEL
LIN {X 0,Y 339.24,Z 579.754,A -85,B 0,C 180,E1 -14908.807,E2 -14908.807} C_VEL
LIN {X 0,Y 339.625,Z 584.125,A -85,B 0,C 180,E1 -14909.88,E2 -14909.88} C_VEL
LIN {X 0,Y 336.704,Z 604.057,A -85,B 0,C 180,E1 -14913.838,E2 -14913.838} C_VEL
LIN {X 0,Y 334.047,Z 625.515,A -85,B 0,C 180,E1 -14918.013,E2 -14918.013} C_VEL
LIN {X 0,Y 333.399,Z 632.565,A -85,B 0,C 180,E1 -14919.324,E2 -14919.324} C_VEL
LIN {X 0,Y 336.12,Z 647.345,A -85,B 0,C 180,E1 -14920.28,E2 -14920.28} C_VEL
LIN {X 0,Y 337.154,Z 656.733,A -85,B 0,C 180,E1 -14920.777,E2 -14920.777} C_VEL
LIN {X 0,Y 334.491,Z 706.022,A -85,B 0,C 180,E1 -14922.46,E2 -14922.46} C_VEL
LIN {X 0,Y 333.663,Z 716.609,A -85,B 0,C 180,E1 -14923.007,E2 -14923.007} C_VEL
LIN {X 0,Y 332.729,Z 726.772,A -85,B 0,C 180,E1 -14923.748,E2 -14923.748} C_VEL
LIN {X 0,Y 331.632,Z 735.952,A -85,B 0,C 180,E1 -14924.639,E2 -14924.639} C_VEL
LIN {X 0,Y 330.53,Z 744.537,A -85,B 0,C 180,E1 -14925.689,E2 -14925.689} C_VEL
LIN {X 0,Y 329.279,Z 753.243,A -85,B 0,C 180,E1 -14927.05,E2 -14927.05} C_VEL
LIN {X 0,Y 328.046,Z 760.878,A -85,B 0,C 180,E1 -14928.57,E2 -14928.57} C_VEL
LIN {X 0,Y 327.09,Z 766.911,A -85,B 0,C 180,E1 -14930.102,E2 -14930.102} C_VEL
LIN {X 0,Y 326.506,Z 770.713,A -85,B 0,C 180,E1 -14931.334,E2 -14931.334} C_VEL
LIN {X 0,Y 326.03,Z 773.763,A -85,B 0,C 180,E1 -14932.569,E2 -14932.569} C_VEL
LIN {X 0,Y 325.726,Z 776.117,A -85,B 0,C 180,E1 -14933.807,E2 -14933.807} C_VEL
LIN {X 0,Y 325.325,Z 777.835,A -85,B 0,C 180,E1 -14935.043,E2 -14935.043} C_VEL
LIN {X 0,Y 325.046,Z 778.95,A -85,B 0,C 180,E1 -14936.281,E2 -14936.281} C_VEL
LIN {X 0,Y 324.885,Z 779.481,A -85,B 0,C 180,E1 -14937.52,E2 -14937.52} C_VEL
LIN {X 0,Y 324.798,Z 779.427,A -85,B 0,C 180,E1 -14938.76,E2 -14938.76} C_VEL
LIN {X 0,Y 324.793,Z 778.789,A -85,B 0,C 180,E1 -14940,E2 -14940} C_VEL
LIN {X 0,Y 324.79,Z 777.554,A -85,B 0,C 180,E1 -14941.24,E2 -14941.24} C_VEL
LIN {X 0,Y 324.921,Z 774.505,A -85,B 0,C 180,E1 -14943.1,E2 -14943.1} C_VEL
LIN {X 0,Y 325.054,Z 771.627,A -85,B 0,C 180,E1 -14944.34,E2 -14944.34} C_VEL
LIN {X 0,Y 325.15,Z 766.176,A -85,B 0,C 180,E1 -14946.129,E2 -14946.129} C_VEL
LIN {X 0,Y 325.48,Z 760.921,A -85,B 0,C 180,E1 -14947.444,E2 -14947.444} C_VEL
LIN {X 0,Y 325.773,Z 754.833,A -85,B 0,C 180,E1 -14948.686,E2 -14948.686} C_VEL
LIN {X 0,Y 326.197,Z 747.401,A -85,B 0,C 180,E1 -14949.925,E2 -14949.925} C_VEL
LIN {X 0,Y 326.651,Z 738.008,A -85,B 0,C 180,E1 -14951.165,E2 -14951.165} C_VEL
LIN {X 0,Y 327.143,Z 728.914,A -85,B 0,C 180,E1 -14952.091,E2 -14952.091} C_VEL
LIN {X 0,Y 327.556,Z 718.091,A -85,B 0,C 180,E1 -14952.941,E2 -14952.941} C_VEL
LIN {X 0,Y 328.01,Z 707.385,A -85,B 0,C 180,E1 -14953.514,E2 -14953.514} C_VEL
LIN {X 0,Y 328.242,Z 693.968,A -85,B 0,C 180,E1 -14953.978,E2 -14953.978} C_VEL
LIN {X 0,Y 329.085,Z 651.93,A -85,B 0,C 180,E1 -14955.244,E2 -14955.244} C_VEL
LIN {X 0,Y 327.489,Z 631.769,A -85,B 0,C 180,E1 -14955.935,E2 -14955.935} C_VEL
LIN {X 0,Y 328.498,Z 613.461,A -85,B 0,C 180,E1 -14959.288,E2 -14959.288} C_VEL
LIN {X 0,Y 329.75,Z 594.032,A -85,B 0,C 180,E1 -14962.865,E2 -14962.865} C_VEL
LIN {X 0,Y 331.309,Z 571.588,A -85,B 0,C 180,E1 -14967.007,E2 -14967.007} C_VEL
LIN {X 0,Y 331.49,Z 567.315,A -85,B 0,C 180,E1 -14967.803,E2 -14967.803} C_VEL
LIN {X 0,Y 329.192,Z 555.673,A -85,B 0,C 180,E1 -14970.113,E2 -14970.113} C_VEL
LIN {X 0,Y 326.65,Z 543.968,A -85,B 0,C 180,E1 -14972.54,E2 -14972.54} C_VEL
LIN {X 0,Y 326.617,Z 543.8,A -85,B 0,C 180,E1 -14975.519,E2 -14975.519} C_VEL
LIN {X 0,Y 326.616,Z 543.796,A -85,B 0,C 180,E1 -14979.227,E2 -14979.227} C_VEL
LIN {X 0,Y 326.586,Z 543.761,A -85,B 0,C 180,E1 -14982.973,E2 -14982.973} C_VEL
LIN {X 0,Y 326.614,Z 543.8,A -85,B 0,C 180,E1 -14987.021,E2 -14987.021} C_VEL
LIN {X 0,Y 326.616,Z 543.772,A -85,B 0,C 180,E1 -14990.772,E2 -14990.772} C_VEL
LIN {X 0,Y 326.617,Z 543.794,A -85,B 0,C 180,E1 -14994.48,E2 -14994.48} C_VEL
LIN {X 0,Y 326.612,Z 543.801,A -85,B 0,C 180,E1 -14997.455,E2 -14997.455} C_VEL
LIN {X 0,Y 326.665,Z 543.797,A -85,B 0,C 180,E1 -15000.34,E2 -15000.34} C_VEL
LIN {X 0,Y 326.73,Z 544,A -85,B 0,C 180,E1 -15002.315,E2 -15002.315} C_VEL
LIN {X 0,Y 328.6,Z 552.915,A -85,B 0,C 180,E1 -15005.304,E2 -15005.304} C_VEL
LIN {X 0,Y 329.022,Z 554.369,A -85,B 0,C 180,E1 -15005.473,E2 -15005.473} C_VEL
LIN {X 0,Y 335.126,Z 570.282,A -85,B 0,C 180,E1 -15006.329,E2 -15006.329} C_VEL
LIN {X 0,Y 337.718,Z 583.713,A -85,B 0,C 180,E1 -15006.829,E2 -15006.829} C_VEL
LIN {X 0,Y 336.018,Z 659.531,A -85,B 0,C 180,E1 -15008.448,E2 -15008.448} C_VEL
LIN {X 0,Y 335.384,Z 672.948,A -85,B 0,C 180,E1 -15008.969,E2 -15008.969} C_VEL
LIN {X 0,Y 334.513,Z 685.715,A -85,B 0,C 180,E1 -15009.716,E2 -15009.716} C_VEL
LIN {X 0,Y 333.436,Z 697.042,A -85,B 0,C 180,E1 -15010.611,E2 -15010.611} C_VEL
LIN {X 0,Y 332.051,Z 708.949,A -85,B 0,C 180,E1 -15011.84,E2 -15011.84} C_VEL
LIN {X 0,Y 330.918,Z 719.38,A -85,B 0,C 180,E1 -15013.215,E2 -15013.215} C_VEL
LIN {X 0,Y 329.775,Z 727.682,A -85,B 0,C 180,E1 -15014.549,E2 -15014.549} C_VEL
LIN {X 0,Y 328.585,Z 735.551,A -85,B 0,C 180,E1 -15016.076,E2 -15016.076} C_VEL
LIN {X 0,Y 327.425,Z 743.237,A -85,B 0,C 180,E1 -15017.919,E2 -15017.919} C_VEL
LIN {X 0,Y 326.378,Z 750.294,A -85,B 0,C 180,E1 -15020.079,E2 -15020.079} C_VEL
LIN {X 0,Y 325.765,Z 754.991,A -85,B 0,C 180,E1 -15021.938,E2 -15021.938} C_VEL
LIN {X 0,Y 325.388,Z 758.579,A -85,B 0,C 180,E1 -15023.799,E2 -15023.799} C_VEL
LIN {X 0,Y 325.229,Z 760.434,A -85,B 0,C 180,E1 -15025.04,E2 -15025.04} C_VEL
LIN {X 0,Y 325.056,Z 761.832,A -85,B 0,C 180,E1 -15026.28,E2 -15026.28} C_VEL
LIN {X 0,Y 324.876,Z 763.44,A -85,B 0,C 180,E1 -15028.759,E2 -15028.759} C_VEL
LIN {X 0,Y 324.88,Z 763.672,A -85,B 0,C 180,E1 -15029.999,E2 -15029.999} C_VEL
LIN {X 0,Y 324.876,Z 763.482,A -85,B 0,C 180,E1 -15031.238,E2 -15031.238} C_VEL
LIN {X 0,Y 325.051,Z 761.932,A -85,B 0,C 180,E1 -15033.718,E2 -15033.718} C_VEL
LIN {X 0,Y 325.223,Z 760.576,A -85,B 0,C 180,E1 -15034.958,E2 -15034.958} C_VEL
LIN {X 0,Y 325.449,Z 758.076,A -85,B 0,C 180,E1 -15036.604,E2 -15036.604} C_VEL
LIN {X 0,Y 325.906,Z 753.822,A -85,B 0,C 180,E1 -15038.681,E2 -15038.681} C_VEL
LIN {X 0,Y 326.657,Z 748.806,A -85,B 0,C 180,E1 -15040.536,E2 -15040.536} C_VEL
LIN {X 0,Y 327.567,Z 742.491,A -85,B 0,C 180,E1 -15042.388,E2 -15042.388} C_VEL
LIN {X 0,Y 328.668,Z 734.585,A -85,B 0,C 180,E1 -15044.234,E2 -15044.234} C_VEL
LIN {X 0,Y 330.266,Z 724.743,A -85,B 0,C 180,E1 -15046.058,E2 -15046.058} C_VEL
LIN {X 0,Y 331.494,Z 714.418,A -85,B 0,C 180,E1 -15047.583,E2 -15047.583} C_VEL
LIN {X 0,Y 332.643,Z 704.192,A -85,B 0,C 180,E1 -15048.795,E2 -15048.795} C_VEL
LIN {X 0,Y 333.885,Z 692.988,A -85,B 0,C 180,E1 -15049.84,E2 -15049.84} C_VEL
LIN {X 0,Y 335.002,Z 680.354,A -85,B 0,C 180,E1 -15050.732,E2 -15050.732} C_VEL
LIN {X 0,Y 335.731,Z 667.7,A -85,B 0,C 180,E1 -15051.368,E2 -15051.368} C_VEL
LIN {X 0,Y 336.291,Z 654.679,A -85,B 0,C 180,E1 -15051.773,E2 -15051.773} C_VEL
LIN {X 0,Y 337.114,Z 614.656,A -85,B 0,C 180,E1 -15052.622,E2 -15052.622} C_VEL
LIN {X 0,Y 336.337,Z 606.962,A -85,B 0,C 180,E1 -15052.852,E2 -15052.852} C_VEL
LIN {X 0,Y 332.556,Z 592.022,A -85,B 0,C 180,E1 -15053.474,E2 -15053.474} C_VEL
LIN {X 0,Y 331.166,Z 584.402,A -85,B 0,C 180,E1 -15053.757,E2 -15053.757} C_VEL
LIN {X 0,Y 328.487,Z 571.098,A -85,B 0,C 180,E1 -15054.277,E2 -15054.277} C_VEL
LIN {X 0,Y 321.584,Z 553.759,A -85,B 0,C 180,E1 -15055.289,E2 -15055.289} C_VEL
LIN {X 0,Y 321.241,Z 552.289,A -85,B 0,C 180,E1 -15055.653,E2 -15055.653} C_VEL
LIN {X 0,Y 319.637,Z 544.818,A -85,B 0,C 180,E1 -15058.281,E2 -15058.281} C_VEL
LIN {X 0,Y 319.53,Z 544.683,A -85,B 0,C 180,E1 -15061.86,E2 -15061.86} C_VEL
LIN {X 0,Y 319.578,Z 544.671,A -85,B 0,C 180,E1 -15065.542,E2 -15065.542} C_VEL
LIN {X 0,Y 319.578,Z 544.677,A -85,B 0,C 180,E1 -15068.006,E2 -15068.006} C_VEL
LIN {X 0,Y 319.525,Z 544.684,A -85,B 0,C 180,E1 -15071.596,E2 -15071.596} C_VEL
LIN {X 0,Y 319.489,Z 544.671,A -85,B 0,C 180,E1 -15075.257,E2 -15075.257} C_VEL
LIN {X 0,Y 319.564,Z 544.677,A -85,B 0,C 180,E1 -15078.393,E2 -15078.393} C_VEL
LIN {X 0,Y 319.578,Z 544.657,A -85,B 0,C 180,E1 -15082.342,E2 -15082.342} C_VEL
LIN {X 0,Y 319.561,Z 544.68,A -85,B 0,C 180,E1 -15085.123,E2 -15085.123} C_VEL
LIN {X 0,Y 319.564,Z 544.676,A -85,B 0,C 180,E1 -15089.057,E2 -15089.057} C_VEL
LIN {X 0,Y 319.602,Z 544.662,A -85,B 0,C 180,E1 -15092.497,E2 -15092.497} C_VEL
LIN {X 0,Y 319.599,Z 544.676,A -85,B 0,C 180,E1 -15095.303,E2 -15095.303} C_VEL
LIN {X 0,Y 319.59,Z 544.664,A -85,B 0,C 180,E1 -15098.047,E2 -15098.047} C_VEL
LIN {X 0,Y 319.682,Z 544.662,A -85,B 0,C 180,E1 -15100.961,E2 -15100.961} C_VEL
LIN {X 0,Y 319.723,Z 544.651,A -85,B 0,C 180,E1 -15105.275,E2 -15105.275} C_VEL
LIN {X 0,Y 319.75,Z 544.641,A -85,B 0,C 180,E1 -15109.873,E2 -15109.873} C_VEL
LIN {X 0,Y 319.926,Z 544.63,A -85,B 0,C 180,E1 -15112.426,E2 -15112.426} C_VEL
LIN {X 0,Y 319.742,Z 544.654,A -85,B 0,C 180,E1 -15114.956,E2 -15114.956} C_VEL
LIN {X 0,Y 319.984,Z 544.613,A -85,B 0,C 180,E1 -15117.482,E2 -15117.482} C_VEL
LIN {X 0,Y 320.162,Z 544.604,A -85,B 0,C 180,E1 -15120,E2 -15120} C_VEL
LIN {X 0,Y 319.985,Z 544.617,A -85,B 0,C 180,E1 -15122.518,E2 -15122.518} C_VEL
LIN {X 0,Y 319.947,Z 544.629,A -85,B 0,C 180,E1 -15126.306,E2 -15126.306} C_VEL
LIN {X 0,Y 319.835,Z 544.639,A -85,B 0,C 180,E1 -15128.848,E2 -15128.848} C_VEL
LIN {X 0,Y 319.677,Z 544.662,A -85,B 0,C 180,E1 -15132.7,E2 -15132.7} C_VEL
LIN {X 0,Y 319.692,Z 544.655,A -85,B 0,C 180,E1 -15135.296,E2 -15135.296} C_VEL
LIN {X 0,Y 319.67,Z 544.666,A -85,B 0,C 180,E1 -15139.255,E2 -15139.255} C_VEL
LIN {X 0,Y 319.564,Z 544.675,A -85,B 0,C 180,E1 -15143.32,E2 -15143.32} C_VEL
LIN {X 0,Y 319.611,Z 544.664,A -85,B 0,C 180,E1 -15146.09,E2 -15146.09} C_VEL
LIN {X 0,Y 319.573,Z 544.677,A -85,B 0,C 180,E1 -15148.935,E2 -15148.935} C_VEL
LIN {X 0,Y 319.525,Z 544.681,A -85,B 0,C 180,E1 -15151.863,E2 -15151.863} C_VEL
LIN {X 0,Y 319.574,Z 544.659,A -85,B 0,C 180,E1 -15155.544,E2 -15155.544} C_VEL
LIN {X 0,Y 319.552,Z 544.668,A -85,B 0,C 180,E1 -15158.011,E2 -15158.011} C_VEL
LIN {X 0,Y 319.549,Z 544.669,A -85,B 0,C 180,E1 -15161.604,E2 -15161.604} C_VEL
LIN {X 0,Y 319.575,Z 544.679,A -85,B 0,C 180,E1 -15165.275,E2 -15165.275} C_VEL
LIN {X 0,Y 319.575,Z 544.677,A -85,B 0,C 180,E1 -15168.721,E2 -15168.721} C_VEL
LIN {X 0,Y 319.579,Z 544.645,A -85,B 0,C 180,E1 -15172.344,E2 -15172.344} C_VEL
LIN {X 0,Y 319.558,Z 544.68,A -85,B 0,C 180,E1 -15175.125,E2 -15175.125} C_VEL
LIN {X 0,Y 319.584,Z 544.79,A -85,B 0,C 180,E1 -15177.401,E2 -15177.401} C_VEL
LIN {X 0,Y 322.042,Z 555.478,A -85,B 0,C 180,E1 -15180.801,E2 -15180.801} C_VEL
LIN {X 0,Y 323.868,Z 564.77,A -85,B 0,C 180,E1 -15183.587,E2 -15183.587} C_VEL
LIN {X 0,Y 324.192,Z 568.983,A -85,B 0,C 180,E1 -15184.771,E2 -15184.771} C_VEL
LIN {X 0,Y 324.128,Z 570.025,A -85,B 0,C 180,E1 -15184.956,E2 -15184.956} C_VEL
LIN {X 0,Y 329.015,Z 597.523,A -85,B 0,C 180,E1 -15186.023,E2 -15186.023} C_VEL
LIN {X 0,Y 330.742,Z 610.319,A -85,B 0,C 180,E1 -15186.452,E2 -15186.452} C_VEL
LIN {X 0,Y 329.248,Z 678.075,A -85,B 0,C 180,E1 -15187.943,E2 -15187.943} C_VEL
LIN {X 0,Y 328.345,Z 691.246,A -85,B 0,C 180,E1 -15188.457,E2 -15188.457} C_VEL
LIN {X 0,Y 327.379,Z 703.364,A -85,B 0,C 180,E1 -15189.174,E2 -15189.174} C_VEL
LIN {X 0,Y 326.067,Z 715.605,A -85,B 0,C 180,E1 -15190.157,E2 -15190.157} C_VEL
LIN {X 0,Y 324.592,Z 727.182,A -85,B 0,C 180,E1 -15191.377,E2 -15191.377} C_VEL
LIN {X 0,Y 323.153,Z 737.611,A -85,B 0,C 180,E1 -15192.765,E2 -15192.765} C_VEL
LIN {X 0,Y 321.987,Z 746.455,A -85,B 0,C 180,E1 -15194.226,E2 -15194.226} C_VEL
LIN {X 0,Y 320.653,Z 755.388,A -85,B 0,C 180,E1 -15196.05,E2 -15196.05} C_VEL
LIN {X 0,Y 319.501,Z 762.82,A -85,B 0,C 180,E1 -15197.939,E2 -15197.939} C_VEL
LIN {X 0,Y 318.744,Z 768.792,A -85,B 0,C 180,E1 -15199.842,E2 -15199.842} C_VEL
LIN {X 0,Y 318.229,Z 773.514,A -85,B 0,C 180,E1 -15201.748,E2 -15201.748} C_VEL
LIN {X 0,Y 317.89,Z 777.127,A -85,B 0,C 180,E1 -15203.655,E2 -15203.655} C_VEL
LIN {X 0,Y 317.804,Z 778.99,A -85,B 0,C 180,E1 -15204.926,E2 -15204.926} C_VEL
LIN {X 0,Y 317.808,Z 780.388,A -85,B 0,C 180,E1 -15206.197,E2 -15206.197} C_VEL
LIN {X 0,Y 317.731,Z 782.101,A -85,B 0,C 180,E1 -15208.734,E2 -15208.734} C_VEL
LIN {X 0,Y 317.744,Z 783.392,A -85,B 0,C 180,E1 -15210.001,E2 -15210.001} C_VEL
LIN {X 0,Y 317.708,Z 784.14,A -85,B 0,C 180,E1 -15211.269,E2 -15211.269} C_VEL
LIN {X 0,Y 317.76,Z 784.3,A -85,B 0,C 180,E1 -15212.536,E2 -15212.536} C_VEL
LIN {X 0,Y 317.857,Z 783.864,A -85,B 0,C 180,E1 -15213.804,E2 -15213.804} C_VEL
LIN {X 0,Y 317.936,Z 782.808,A -85,B 0,C 180,E1 -15215.074,E2 -15215.074} C_VEL
LIN {X 0,Y 318.169,Z 780.017,A -85,B 0,C 180,E1 -15216.979,E2 -15216.979} C_VEL
LIN {X 0,Y 318.634,Z 775.82,A -85,B 0,C 180,E1 -15218.883,E2 -15218.883} C_VEL
LIN {X 0,Y 319.227,Z 769.981,A -85,B 0,C 180,E1 -15220.787,E2 -15220.787} C_VEL
LIN {X 0,Y 319.685,Z 764.975,A -85,B 0,C 180,E1 -15222.056,E2 -15222.056} C_VEL
LIN {X 0,Y 320.309,Z 758.904,A -85,B 0,C 180,E1 -15223.321,E2 -15223.321} C_VEL
LIN {X 0,Y 320.884,Z 753.909,A -85,B 0,C 180,E1 -15224.265,E2 -15224.265} C_VEL
LIN {X 0,Y 322.122,Z 745.292,A -85,B 0,C 180,E1 -15225.961,E2 -15225.961} C_VEL
LIN {X 0,Y 323.391,Z 735.327,A -85,B 0,C 180,E1 -15227.551,E2 -15227.551} C_VEL
LIN {X 0,Y 324.911,Z 724.401,A -85,B 0,C 180,E1 -15228.934,E2 -15228.934} C_VEL
LIN {X 0,Y 326.444,Z 711.931,A -85,B 0,C 180,E1 -15230.15,E2 -15230.15} C_VEL
LIN {X 0,Y 327.661,Z 699.688,A -85,B 0,C 180,E1 -15231.056,E2 -15231.056} C_VEL
LIN {X 0,Y 328.654,Z 687.703,A -85,B 0,C 180,E1 -15231.689,E2 -15231.689} C_VEL
LIN {X 0,Y 329.3,Z 674.547,A -85,B 0,C 180,E1 -15232.138,E2 -15232.138} C_VEL
LIN {X 0,Y 330.538,Z 608.031,A -85,B 0,C 180,E1 -15233.597,E2 -15233.597} C_VEL
LIN {X 0,Y 330.317,Z 605.618,A -85,B 0,C 180,E1 -15233.721,E2 -15233.721} C_VEL
LIN {X 0,Y 331.922,Z 587.68,A -85,B 0,C 180,E1 -15235.668,E2 -15235.668} C_VEL
LIN {X 0,Y 331.713,Z 579.046,A -85,B 0,C 180,E1 -15236.979,E2 -15236.979} C_VEL
LIN {X 0,Y 331.661,Z 577.404,A -85,B 0,C 180,E1 -15237.263,E2 -15237.263} C_VEL
LIN {X 0,Y 329.516,Z 567.201,A -85,B 0,C 180,E1 -15239.705,E2 -15239.705} C_VEL
LIN {X 0,Y 328.436,Z 561.107,A -85,B 0,C 180,E1 -15241.504,E2 -15241.504} C_VEL
LIN {X 0,Y 327.654,Z 558.947,A -85,B 0,C 180,E1 -15242.429,E2 -15242.429} C_VEL
LIN {X 0,Y 325.516,Z 555.24,A -85,B 0,C 180,E1 -15244.872,E2 -15244.872} C_VEL
LIN {X 0,Y 325.023,Z 554.204,A -85,B 0,C 180,E1 -15245.721,E2 -15245.721} C_VEL
LIN {X 0,Y 323.588,Z 552.557,A -85,B 0,C 180,E1 -15248.566,E2 -15248.566} C_VEL
LIN {X 0,Y 323.246,Z 552.192,A -85,B 0,C 180,E1 -15250.713,E2 -15250.713} C_VEL
LIN {X 0,Y 323.368,Z 552.482,A -85,B 0,C 180,E1 -15252.358,E2 -15252.358} C_VEL
LIN {X 0,Y 323.978,Z 553.35,A -85,B 0,C 180,E1 -15254.286,E2 -15254.286} C_VEL
LIN {X 0,Y 324.723,Z 555.09,A -85,B 0,C 180,E1 -15256.165,E2 -15256.165} C_VEL
LIN {X 0,Y 326.379,Z 558.717,A -85,B 0,C 180,E1 -15258.91,E2 -15258.91} C_VEL
LIN {X 0,Y 328.399,Z 563.818,A -85,B 0,C 180,E1 -15261.638,E2 -15261.638} C_VEL
LIN {X 0,Y 330.255,Z 569.308,A -85,B 0,C 180,E1 -15263.966,E2 -15263.966} C_VEL
LIN {X 0,Y 331.848,Z 575.389,A -85,B 0,C 180,E1 -15266.085,E2 -15266.085} C_VEL
LIN {X 0,Y 333.282,Z 582.262,A -85,B 0,C 180,E1 -15268.185,E2 -15268.185} C_VEL
LIN {X 0,Y 333.719,Z 586.383,A -85,B 0,C 180,E1 -15269.292,E2 -15269.292} C_VEL
LIN {X 0,Y 330.974,Z 603.762,A -85,B 0,C 180,E1 -15272.837,E2 -15272.837} C_VEL
LIN {X 0,Y 328.254,Z 623.265,A -85,B 0,C 180,E1 -15276.733,E2 -15276.733} C_VEL
LIN {X 0,Y 327.223,Z 632.422,A -85,B 0,C 180,E1 -15278.502,E2 -15278.502} C_VEL
LIN {X 0,Y 329.867,Z 646.536,A -85,B 0,C 180,E1 -15279.498,E2 -15279.498} C_VEL
LIN {X 0,Y 331.129,Z 656.996,A -85,B 0,C 180,E1 -15280.111,E2 -15280.111} C_VEL
LIN {X 0,Y 328.35,Z 705.945,A -85,B 0,C 180,E1 -15281.839,E2 -15281.839} C_VEL
LIN {X 0,Y 327.426,Z 716.999,A -85,B 0,C 180,E1 -15282.432,E2 -15282.432} C_VEL
LIN {X 0,Y 326.308,Z 727.756,A -85,B 0,C 180,E1 -15283.258,E2 -15283.258} C_VEL
LIN {X 0,Y 325.131,Z 736.769,A -85,B 0,C 180,E1 -15284.163,E2 -15284.163} C_VEL
LIN {X 0,Y 323.819,Z 746.333,A -85,B 0,C 180,E1 -15285.386,E2 -15285.386} C_VEL
LIN {X 0,Y 322.478,Z 754.616,A -85,B 0,C 180,E1 -15286.772,E2 -15286.772} C_VEL
LIN {X 0,Y 321.429,Z 760.62,A -85,B 0,C 180,E1 -15288.011,E2 -15288.011} C_VEL
LIN {X 0,Y 320.371,Z 766.699,A -85,B 0,C 180,E1 -15289.573,E2 -15289.573} C_VEL
LIN {X 0,Y 319.528,Z 771.347,A -85,B 0,C 180,E1 -15291.143,E2 -15291.143} C_VEL
LIN {X 0,Y 319.001,Z 774.442,A -85,B 0,C 180,E1 -15292.488,E2 -15292.488} C_VEL
LIN {X 0,Y 318.7,Z 776.553,A -85,B 0,C 180,E1 -15293.67,E2 -15293.67} C_VEL
LIN {X 0,Y 318.286,Z 778.188,A -85,B 0,C 180,E1 -15294.933,E2 -15294.933} C_VEL
LIN {X 0,Y 317.986,Z 779.2,A -85,B 0,C 180,E1 -15296.198,E2 -15296.198} C_VEL
LIN {X 0,Y 317.809,Z 779.604,A -85,B 0,C 180,E1 -15297.465,E2 -15297.465} C_VEL
LIN {X 0,Y 317.713,Z 779.428,A -85,B 0,C 180,E1 -15298.733,E2 -15298.733} C_VEL
LIN {X 0,Y 317.704,Z 778.673,A -85,B 0,C 180,E1 -15300,E2 -15300} C_VEL
LIN {X 0,Y 317.705,Z 777.32,A -85,B 0,C 180,E1 -15301.268,E2 -15301.268} C_VEL
LIN {X 0,Y 317.853,Z 774.137,A -85,B 0,C 180,E1 -15303.169,E2 -15303.169} C_VEL
LIN {X 0,Y 317.968,Z 771.118,A -85,B 0,C 180,E1 -15304.437,E2 -15304.437} C_VEL
LIN {X 0,Y 318.124,Z 765.087,A -85,B 0,C 180,E1 -15306.342,E2 -15306.342} C_VEL
LIN {X 0,Y 318.426,Z 759.932,A -85,B 0,C 180,E1 -15307.61,E2 -15307.61} C_VEL
LIN {X 0,Y 318.739,Z 753.634,A -85,B 0,C 180,E1 -15308.879,E2 -15308.879} C_VEL
LIN {X 0,Y 319.168,Z 744.788,A -85,B 0,C 180,E1 -15310.306,E2 -15310.306} C_VEL
LIN {X 0,Y 319.68,Z 735.97,A -85,B 0,C 180,E1 -15311.412,E2 -15311.412} C_VEL
LIN {X 0,Y 320.138,Z 726.473,A -85,B 0,C 180,E1 -15312.359,E2 -15312.359} C_VEL
LIN {X 0,Y 320.554,Z 715.713,A -85,B 0,C 180,E1 -15313.148,E2 -15313.148} C_VEL
LIN {X 0,Y 320.994,Z 705.149,A -85,B 0,C 180,E1 -15313.694,E2 -15313.694} C_VEL
LIN {X 0,Y 321.965,Z 651.797,A -85,B 0,C 180,E1 -15315.402,E2 -15315.402} C_VEL
LIN {X 0,Y 320.449,Z 631.86,A -85,B 0,C 180,E1 -15316.09,E2 -15316.09} C_VEL
LIN {X 0,Y 321.66,Z 611.461,A -85,B 0,C 180,E1 -15319.879,E2 -15319.879} C_VEL
LIN {X 0,Y 322.927,Z 591.708,A -85,B 0,C 180,E1 -15323.572,E2 -15323.572} C_VEL
LIN {X 0,Y 324.541,Z 569.065,A -85,B 0,C 180,E1 -15327.812,E2 -15327.812} C_VEL
LIN {X 0,Y 322.72,Z 559.155,A -85,B 0,C 180,E1 -15329.799,E2 -15329.799} C_VEL
LIN {X 0,Y 319.61,Z 544.827,A -85,B 0,C 180,E1 -15332.808,E2 -15332.808} C_VEL
LIN {X 0,Y 319.563,Z 544.681,A -85,B 0,C 180,E1 -15336.427,E2 -15336.427} C_VEL
LIN {X 0,Y 319.563,Z 544.674,A -85,B 0,C 180,E1 -15339.668,E2 -15339.668} C_VEL
LIN {X 0,Y 319.561,Z 544.638,A -85,B 0,C 180,E1 -15343.467,E2 -15343.467} C_VEL
LIN {X 0,Y 319.591,Z 544.675,A -85,B 0,C 180,E1 -15347.022,E2 -15347.022} C_VEL
LIN {X 0,Y 319.551,Z 544.65,A -85,B 0,C 180,E1 -15350.37,E2 -15350.37} C_VEL
LIN {X 0,Y 319.584,Z 544.67,A -85,B 0,C 180,E1 -15354.456,E2 -15354.456} C_VEL
LIN {X 0,Y 319.537,Z 544.678,A -85,B 0,C 180,E1 -15358.138,E2 -15358.138} C_VEL
LIN {X 0,Y 319.659,Z 544.787,A -85,B 0,C 180,E1 -15361.821,E2 -15361.821} C_VEL
LIN {X 0,Y 321.396,Z 552.954,A -85,B 0,C 180,E1 -15364.662,E2 -15364.662} C_VEL
LIN {X 0,Y 321.699,Z 554.099,A -85,B 0,C 180,E1 -15364.856,E2 -15364.856} C_VEL
LIN {X 0,Y 328.748,Z 571.943,A -85,B 0,C 180,E1 -15365.874,E2 -15365.874} C_VEL
LIN {X 0,Y 331.193,Z 584.262,A -85,B 0,C 180,E1 -15366.352,E2 -15366.352} C_VEL
LIN {X 0,Y 329.45,Z 659.752,A -85,B 0,C 180,E1 -15367.996,E2 -15367.996} C_VEL
LIN {X 0,Y 328.791,Z 673.162,A -85,B 0,C 180,E1 -15368.527,E2 -15368.527} C_VEL
LIN {X 0,Y 327.89,Z 685.927,A -85,B 0,C 180,E1 -15369.288,E2 -15369.288} C_VEL
LIN {X 0,Y 326.759,Z 697.252,A -85,B 0,C 180,E1 -15370.198,E2 -15370.198} C_VEL
LIN {X 0,Y 325.342,Z 708.901,A -85,B 0,C 180,E1 -15371.419,E2 -15371.419} C_VEL
LIN {X 0,Y 324.22,Z 718.638,A -85,B 0,C 180,E1 -15372.712,E2 -15372.712} C_VEL
LIN {X 0,Y 322.926,Z 727.89,A -85,B 0,C 180,E1 -15374.213,E2 -15374.213} C_VEL
LIN {X 0,Y 321.694,Z 735.758,A -85,B 0,C 180,E1 -15375.771,E2 -15375.771} C_VEL
LIN {X 0,Y 320.484,Z 743.444,A -85,B 0,C 180,E1 -15377.653,E2 -15377.653} C_VEL
LIN {X 0,Y 319.396,Z 750.5,A -85,B 0,C 180,E1 -15379.86,E2 -15379.86} C_VEL
LIN {X 0,Y 318.741,Z 755.197,A -85,B 0,C 180,E1 -15381.759,E2 -15381.759} C_VEL
LIN {X 0,Y 318.336,Z 758.785,A -85,B 0,C 180,E1 -15383.661,E2 -15383.661} C_VEL
LIN {X 0,Y 318.157,Z 760.639,A -85,B 0,C 180,E1 -15384.93,E2 -15384.93} C_VEL
LIN {X 0,Y 317.991,Z 762.037,A -85,B 0,C 180,E1 -15386.197,E2 -15386.197} C_VEL
LIN {X 0,Y 317.787,Z 763.645,A -85,B 0,C 180,E1 -15388.732,E2 -15388.732} C_VEL
LIN {X 0,Y 317.788,Z 763.877,A -85,B 0,C 180,E1 -15389.999,E2 -15389.999} C_VEL
LIN {X 0,Y 317.787,Z 763.687,A -85,B 0,C 180,E1 -15391.266,E2 -15391.266} C_VEL
LIN {X 0,Y 317.986,Z 762.136,A -85,B 0,C 180,E1 -15393.801,E2 -15393.801} C_VEL
LIN {X 0,Y 318.151,Z 760.78,A -85,B 0,C 180,E1 -15395.068,E2 -15395.068} C_VEL
LIN {X 0,Y 318.385,Z 758.494,A -85,B 0,C 180,E1 -15396.622,E2 -15396.622} C_VEL
LIN {X 0,Y 318.892,Z 754.025,A -85,B 0,C 180,E1 -15398.873,E2 -15398.873} C_VEL
LIN {X 0,Y 319.683,Z 749.009,A -85,B 0,C 180,E1 -15400.769,E2 -15400.769} C_VEL
LIN {X 0,Y 320.621,Z 742.694,A -85,B 0,C 180,E1 -15402.661,E2 -15402.661} C_VEL
LIN {X 0,Y 321.8,Z 734.787,A -85,B 0,C 180,E1 -15404.545,E2 -15404.545} C_VEL
LIN {X 0,Y 323.44,Z 724.945,A -85,B 0,C 180,E1 -15406.407,E2 -15406.407} C_VEL
LIN {X 0,Y 324.728,Z 714.619,A -85,B 0,C 180,E1 -15407.962,E2 -15407.962} C_VEL
LIN {X 0,Y 325.95,Z 704.391,A -85,B 0,C 180,E1 -15409.195,E2 -15409.195} C_VEL
LIN {X 0,Y 327.236,Z 693.186,A -85,B 0,C 180,E1 -15410.261,E2 -15410.261} C_VEL
LIN {X 0,Y 328.383,Z 680.55,A -85,B 0,C 180,E1 -15411.17,E2 -15411.17} C_VEL
LIN {X 0,Y 329.143,Z 667.891,A -85,B 0,C 180,E1 -15411.817,E2 -15411.817} C_VEL
LIN {X 0,Y 329.724,Z 654.862,A -85,B 0,C 180,E1 -15412.229,E2 -15412.229} C_VEL
LIN {X 0,Y 331.166,Z 584.402,A -85,B 0,C 180,E1 -15413.757,E2 -15413.757} C_VEL
LIN {X 0,Y 330.359,Z 580.673,A -85,B 0,C 180,E1 -15413.906,E2 -15413.906} C_VEL
LIN {X 0,Y 328.017,Z 575.54,A -85,B 0,C 180,E1 -15414.209,E2 -15414.209} C_VEL
LIN {X 0,Y 324.887,Z 570.898,A -85,B 0,C 180,E1 -15414.571,E2 -15414.571} C_VEL
LIN {X 0,Y 318.066,Z 561.721,A -85,B 0,C 180,E1 -15415.363,E2 -15415.363} C_VEL
LIN {X 0,Y 316.197,Z 558.365,A -85,B 0,C 180,E1 -15415.608,E2 -15415.608} C_VEL
LIN {X 0,Y 314.353,Z 553.675,A -85,B 0,C 180,E1 -15415.944,E2 -15415.944} C_VEL
LIN {X 0,Y 312.937,Z 547.284,A -85,B 0,C 180,E1 -15418.138,E2 -15418.138} C_VEL
LIN {X 0,Y 312.56,Z 545.563,A -85,B 0,C 180,E1 -15418.859,E2 -15418.859} C_VEL
LIN {X 0,Y 312.502,Z 545.554,A -85,B 0,C 180,E1 -15422.665,E2 -15422.665} C_VEL
LIN {X 0,Y 312.533,Z 545.547,A -85,B 0,C 180,E1 -15425.949,E2 -15425.949} C_VEL
LIN {X 0,Y 312.509,Z 545.55,A -85,B 0,C 180,E1 -15429.025,E2 -15429.025} C_VEL
LIN {X 0,Y 312.488,Z 545.56,A -85,B 0,C 180,E1 -15432.43,E2 -15432.43} C_VEL
LIN {X 0,Y 312.473,Z 545.551,A -85,B 0,C 180,E1 -15436.03,E2 -15436.03} C_VEL
LIN {X 0,Y 312.496,Z 545.551,A -85,B 0,C 180,E1 -15439.292,E2 -15439.292} C_VEL
LIN {X 0,Y 312.537,Z 545.537,A -85,B 0,C 180,E1 -15442.616,E2 -15442.616} C_VEL
LIN {X 0,Y 312.515,Z 545.554,A -85,B 0,C 180,E1 -15446.31,E2 -15446.31} C_VEL
LIN {X 0,Y 312.54,Z 545.552,A -85,B 0,C 180,E1 -15450.349,E2 -15450.349} C_VEL
LIN {X 0,Y 312.596,Z 545.546,A -85,B 0,C 180,E1 -15454.064,E2 -15454.064} C_VEL
LIN {X 0,Y 312.58,Z 545.538,A -85,B 0,C 180,E1 -15457.528,E2 -15457.528} C_VEL
LIN {X 0,Y 312.631,Z 545.539,A -85,B 0,C 180,E1 -15461.656,E2 -15461.656} C_VEL
LIN {X 0,Y 312.686,Z 545.532,A -85,B 0,C 180,E1 -15465.686,E2 -15465.686} C_VEL
LIN {X 0,Y 312.694,Z 545.521,A -85,B 0,C 180,E1 -15469.641,E2 -15469.641} C_VEL
LIN {X 0,Y 312.864,Z 545.51,A -85,B 0,C 180,E1 -15472.254,E2 -15472.254} C_VEL
LIN {X 0,Y 312.712,Z 545.529,A -85,B 0,C 180,E1 -15474.842,E2 -15474.842} C_VEL
LIN {X 0,Y 312.985,Z 545.492,A -85,B 0,C 180,E1 -15478.713,E2 -15478.713} C_VEL
LIN {X 0,Y 313.114,Z 545.482,A -85,B 0,C 180,E1 -15480,E2 -15480} C_VEL
LIN {X 0,Y 312.931,Z 545.496,A -85,B 0,C 180,E1 -15482.574,E2 -15482.574} C_VEL
LIN {X 0,Y 312.905,Z 545.506,A -85,B 0,C 180,E1 -15486.448,E2 -15486.448} C_VEL
LIN {X 0,Y 312.78,Z 545.517,A -85,B 0,C 180,E1 -15489.049,E2 -15489.049} C_VEL
LIN {X 0,Y 312.629,Z 545.54,A -85,B 0,C 180,E1 -15492.991,E2 -15492.991} C_VEL
LIN {X 0,Y 312.631,Z 545.531,A -85,B 0,C 180,E1 -15495.65,E2 -15495.65} C_VEL
LIN {X 0,Y 312.6,Z 545.545,A -85,B 0,C 180,E1 -15499.709,E2 -15499.709} C_VEL
LIN {X 0,Y 312.539,Z 545.548,A -85,B 0,C 180,E1 -15502.79,E2 -15502.79} C_VEL
LIN {X 0,Y 312.59,Z 545.54,A -85,B 0,C 180,E1 -15505.934,E2 -15505.934} C_VEL
LIN {X 0,Y 312.531,Z 545.554,A -85,B 0,C 180,E1 -15509.651,E2 -15509.651} C_VEL
LIN {X 0,Y 312.513,Z 545.556,A -85,B 0,C 180,E1 -15513.69,E2 -15513.69} C_VEL
LIN {X 0,Y 312.52,Z 545.535,A -85,B 0,C 180,E1 -15517.386,E2 -15517.386} C_VEL
LIN {X 0,Y 312.486,Z 545.558,A -85,B 0,C 180,E1 -15520.71,E2 -15520.71} C_VEL
LIN {X 0,Y 312.519,Z 545.555,A -85,B 0,C 180,E1 -15524.198,E2 -15524.198} C_VEL
LIN {X 0,Y 312.544,Z 545.546,A -85,B 0,C 180,E1 -15527.907,E2 -15527.907} C_VEL
LIN {X 0,Y 312.541,Z 545.521,A -85,B 0,C 180,E1 -15531.909,E2 -15531.909} C_VEL
LIN {X 0,Y 312.504,Z 545.536,A -85,B 0,C 180,E1 -15535.791,E2 -15535.791} C_VEL
LIN {X 0,Y 312.566,Z 545.684,A -85,B 0,C 180,E1 -15536.913,E2 -15536.913} C_VEL
LIN {X 0,Y 315.147,Z 557.047,A -85,B 0,C 180,E1 -15540.621,E2 -15540.621} C_VEL
LIN {X 0,Y 317.089,Z 567.048,A -85,B 0,C 180,E1 -15543.688,E2 -15543.688} C_VEL
LIN {X 0,Y 317.339,Z 569.659,A -85,B 0,C 180,E1 -15544.371,E2 -15544.371} C_VEL
LIN {X 0,Y 320.424,Z 586.153,A -85,B 0,C 180,E1 -15545.07,E2 -15545.07} C_VEL
LIN {X 0,Y 324.173,Z 609.793,A -85,B 0,C 180,E1 -15545.937,E2 -15545.937} C_VEL
LIN {X 0,Y 322.653,Z 677.883,A -85,B 0,C 180,E1 -15547.468,E2 -15547.468} C_VEL
LIN {X 0,Y 321.764,Z 691.05,A -85,B 0,C 180,E1 -15547.994,E2 -15547.994} C_VEL
LIN {X 0,Y 320.751,Z 703.166,A -85,B 0,C 180,E1 -15548.723,E2 -15548.723} C_VEL
LIN {X 0,Y 319.385,Z 715.404,A -85,B 0,C 180,E1 -15549.723,E2 -15549.723} C_VEL
LIN {X 0,Y 317.853,Z 726.98,A -85,B 0,C 180,E1 -15550.967,E2 -15550.967} C_VEL
LIN {X 0,Y 316.35,Z 737.405,A -85,B 0,C 180,E1 -15552.382,E2 -15552.382} C_VEL
LIN {X 0,Y 315.095,Z 746.597,A -85,B 0,C 180,E1 -15553.939,E2 -15553.939} C_VEL
LIN {X 0,Y 313.733,Z 755.184,A -85,B 0,C 180,E1 -15555.736,E2 -15555.736} C_VEL
LIN {X 0,Y 312.532,Z 762.616,A -85,B 0,C 180,E1 -15557.666,E2 -15557.666} C_VEL
LIN {X 0,Y 311.716,Z 768.588,A -85,B 0,C 180,E1 -15559.61,E2 -15559.61} C_VEL
LIN {X 0,Y 311.191,Z 773.31,A -85,B 0,C 180,E1 -15561.56,E2 -15561.56} C_VEL
LIN {X 0,Y 310.821,Z 776.922,A -85,B 0,C 180,E1 -15563.51,E2 -15563.51} C_VEL
LIN {X 0,Y 310.708,Z 778.785,A -85,B 0,C 180,E1 -15564.81,E2 -15564.81} C_VEL
LIN {X 0,Y 310.718,Z 780.183,A -85,B 0,C 180,E1 -15566.11,E2 -15566.11} C_VEL
LIN {X 0,Y 310.682,Z 781.179,A -85,B 0,C 180,E1 -15567.408,E2 -15567.408} C_VEL
LIN {X 0,Y 310.646,Z 781.8,A -85,B 0,C 180,E1 -15568.705,E2 -15568.705} C_VEL
LIN {X 0,Y 310.656,Z 783.131,A -85,B 0,C 180,E1 -15570.001,E2 -15570.001} C_VEL
LIN {X 0,Y 310.624,Z 784.013,A -85,B 0,C 180,E1 -15571.298,E2 -15571.298} C_VEL
LIN {X 0,Y 310.685,Z 784.287,A -85,B 0,C 180,E1 -15572.594,E2 -15572.594} C_VEL
LIN {X 0,Y 310.772,Z 783.931,A -85,B 0,C 180,E1 -15573.891,E2 -15573.891} C_VEL
LIN {X 0,Y 310.855,Z 782.96,A -85,B 0,C 180,E1 -15575.19,E2 -15575.19} C_VEL
LIN {X 0,Y 311.13,Z 780.439,A -85,B 0,C 180,E1 -15577.138,E2 -15577.138} C_VEL
LIN {X 0,Y 311.454,Z 777.966,A -85,B 0,C 180,E1 -15578.435,E2 -15578.435} C_VEL
LIN {X 0,Y 311.88,Z 774.786,A -85,B 0,C 180,E1 -15579.731,E2 -15579.731} C_VEL
LIN {X 0,Y 312.429,Z 769.684,A -85,B 0,C 180,E1 -15581.353,E2 -15581.353} C_VEL
LIN {X 0,Y 313.122,Z 763.269,A -85,B 0,C 180,E1 -15582.972,E2 -15582.972} C_VEL
LIN {X 0,Y 314.131,Z 755.169,A -85,B 0,C 180,E1 -15584.579,E2 -15584.579} C_VEL
LIN {X 0,Y 314.835,Z 747.911,A -85,B 0,C 180,E1 -15585.794,E2 -15585.794} C_VEL
LIN {X 0,Y 316.156,Z 738.314,A -85,B 0,C 180,E1 -15587.465,E2 -15587.465} C_VEL
LIN {X 0,Y 317.646,Z 728.101,A -85,B 0,C 180,E1 -15588.881,E2 -15588.881} C_VEL
LIN {X 0,Y 319.156,Z 716.774,A -85,B 0,C 180,E1 -15590.126,E2 -15590.126} C_VEL
LIN {X 0,Y 320.504,Z 705.033,A -85,B 0,C 180,E1 -15591.128,E2 -15591.128} C_VEL
LIN {X 0,Y 321.647,Z 692.175,A -85,B 0,C 180,E1 -15591.933,E2 -15591.933} C_VEL
LIN {X 0,Y 322.592,Z 678.409,A -85,B 0,C 180,E1 -15592.497,E2 -15592.497} C_VEL
LIN {X 0,Y 324.142,Z 612.333,A -85,B 0,C 180,E1 -15594.009,E2 -15594.009} C_VEL
LIN {X 0,Y 324.838,Z 607.649,A -85,B 0,C 180,E1 -15594.426,E2 -15594.426} C_VEL
LIN {X 0,Y 326.74,Z 590.833,A -85,B 0,C 180,E1 -15596.321,E2 -15596.321} C_VEL
LIN {X 0,Y 326.762,Z 584.25,A -85,B 0,C 180,E1 -15597.338,E2 -15597.338} C_VEL
LIN {X 0,Y 326.752,Z 582.392,A -85,B 0,C 180,E1 -15597.64,E2 -15597.64} C_VEL
LIN {X 0,Y 325.383,Z 574.879,A -85,B 0,C 180,E1 -15599.404,E2 -15599.404} C_VEL
LIN {X 0,Y 324.281,Z 567.913,A -85,B 0,C 180,E1 -15601.343,E2 -15601.343} C_VEL
LIN {X 0,Y 323.849,Z 565.429,A -85,B 0,C 180,E1 -15602.182,E2 -15602.182} C_VEL
LIN {X 0,Y 321.595,Z 561.522,A -85,B 0,C 180,E1 -15604.625,E2 -15604.625} C_VEL
LIN {X 0,Y 320.868,Z 559.917,A -85,B 0,C 180,E1 -15605.863,E2 -15605.863} C_VEL
LIN {X 0,Y 319.624,Z 558.569,A -85,B 0,C 180,E1 -15608.002,E2 -15608.002} C_VEL
LIN {X 0,Y 319.131,Z 558.013,A -85,B 0,C 180,E1 -15609.692,E2 -15609.692} C_VEL
LIN {X 0,Y 318.98,Z 557.963,A -85,B 0,C 180,E1 -15611.486,E2 -15611.486} C_VEL
LIN {X 0,Y 319.28,Z 558.501,A -85,B 0,C 180,E1 -15613.415,E2 -15613.415} C_VEL
LIN {X 0,Y 319.9,Z 559.734,A -85,B 0,C 180,E1 -15615.33,E2 -15615.33} C_VEL
LIN {X 0,Y 321.151,Z 562.866,A -85,B 0,C 180,E1 -15618.079,E2 -15618.079} C_VEL
LIN {X 0,Y 322.871,Z 567.487,A -85,B 0,C 180,E1 -15620.858,E2 -15620.858} C_VEL
LIN {X 0,Y 324.561,Z 572.613,A -85,B 0,C 180,E1 -15623.246,E2 -15623.246} C_VEL
LIN {X 0,Y 326.396,Z 579.924,A -85,B 0,C 180,E1 -15625.956,E2 -15625.956} C_VEL
LIN {X 0,Y 327.555,Z 586.215,A -85,B 0,C 180,E1 -15627.936,E2 -15627.936} C_VEL
LIN {X 0,Y 327.794,Z 590.414,A -85,B 0,C 180,E1 -15629.051,E2 -15629.051} C_VEL
LIN {X 0,Y 324.139,Z 611.596,A -85,B 0,C 180,E1 -15633.449,E2 -15633.449} C_VEL
LIN {X 0,Y 321.2,Z 632.505,A -85,B 0,C 180,E1 -15637.652,E2 -15637.652} C_VEL
LIN {X 0,Y 323.76,Z 646.01,A -85,B 0,C 180,E1 -15638.679,E2 -15638.679} C_VEL
LIN {X 0,Y 325.271,Z 657.82,A -85,B 0,C 180,E1 -15639.414,E2 -15639.414} C_VEL
LIN {X 0,Y 322.204,Z 706.925,A -85,B 0,C 180,E1 -15641.232,E2 -15641.232} C_VEL
LIN {X 0,Y 321.234,Z 717.737,A -85,B 0,C 180,E1 -15641.834,E2 -15641.834} C_VEL
LIN {X 0,Y 320.146,Z 727.475,A -85,B 0,C 180,E1 -15642.596,E2 -15642.596} C_VEL
LIN {X 0,Y 318.904,Z 736.481,A -85,B 0,C 180,E1 -15643.517,E2 -15643.517} C_VEL
LIN {X 0,Y 317.622,Z 744.949,A -85,B 0,C 180,E1 -15644.602,E2 -15644.602} C_VEL
LIN {X 0,Y 316.331,Z 752.712,A -85,B 0,C 180,E1 -15645.854,E2 -15645.854} C_VEL
LIN {X 0,Y 315.129,Z 759.027,A -85,B 0,C 180,E1 -15647.114,E2 -15647.114} C_VEL
LIN {X 0,Y 313.868,Z 765.424,A -85,B 0,C 180,E1 -15648.701,E2 -15648.701} C_VEL
LIN {X 0,Y 312.896,Z 770.461,A -85,B 0,C 180,E1 -15650.302,E2 -15650.302} C_VEL
LIN {X 0,Y 312.007,Z 774.821,A -85,B 0,C 180,E1 -15652.233,E2 -15652.233} C_VEL
LIN {X 0,Y 311.651,Z 776.94,A -85,B 0,C 180,E1 -15653.526,E2 -15653.526} C_VEL
LIN {X 0,Y 311.227,Z 778.471,A -85,B 0,C 180,E1 -15654.818,E2 -15654.818} C_VEL
LIN {X 0,Y 310.929,Z 779.403,A -85,B 0,C 180,E1 -15656.112,E2 -15656.112} C_VEL
LIN {X 0,Y 310.735,Z 779.72,A -85,B 0,C 180,E1 -15657.407,E2 -15657.407} C_VEL
LIN {X 0,Y 310.63,Z 779.422,A -85,B 0,C 180,E1 -15658.704,E2 -15658.704} C_VEL
LIN {X 0,Y 310.618,Z 778.533,A -85,B 0,C 180,E1 -15660,E2 -15660} C_VEL
LIN {X 0,Y 310.647,Z 776.134,A -85,B 0,C 180,E1 -15661.945,E2 -15661.945} C_VEL
LIN {X 0,Y 310.787,Z 773.711,A -85,B 0,C 180,E1 -15663.241,E2 -15663.241} C_VEL
LIN {X 0,Y 310.884,Z 770.57,A -85,B 0,C 180,E1 -15664.538,E2 -15664.538} C_VEL
LIN {X 0,Y 311.077,Z 764.269,A -85,B 0,C 180,E1 -15666.486,E2 -15666.486} C_VEL
LIN {X 0,Y 311.437,Z 757.474,A -85,B 0,C 180,E1 -15668.108,E2 -15668.108} C_VEL
LIN {X 0,Y 311.859,Z 749.529,A -85,B 0,C 180,E1 -15669.567,E2 -15669.567} C_VEL
LIN {X 0,Y 312.229,Z 741.89,A -85,B 0,C 180,E1 -15670.702,E2 -15670.702} C_VEL
LIN {X 0,Y 312.838,Z 732.455,A -85,B 0,C 180,E1 -15671.829,E2 -15671.829} C_VEL
LIN {X 0,Y 313.284,Z 722.583,A -85,B 0,C 180,E1 -15672.717,E2 -15672.717} C_VEL
LIN {X 0,Y 313.597,Z 713.178,A -85,B 0,C 180,E1 -15673.363,E2 -15673.363} C_VEL
LIN {X 0,Y 313.988,Z 701.212,A -85,B 0,C 180,E1 -15673.923,E2 -15673.923} C_VEL
LIN {X 0,Y 314.955,Z 652.721,A -85,B 0,C 180,E1 -15675.498,E2 -15675.498} C_VEL
LIN {X 0,Y 313.4,Z 632.126,A -85,B 0,C 180,E1 -15676.237,E2 -15676.237} C_VEL
LIN {X 0,Y 313.837,Z 624.66,A -85,B 0,C 180,E1 -15677.597,E2 -15677.597} C_VEL
LIN {X 0,Y 315.138,Z 603.614,A -85,B 0,C 180,E1 -15681.591,E2 -15681.591} C_VEL
LIN {X 0,Y 316.504,Z 584.058,A -85,B 0,C 180,E1 -15685.306,E2 -15685.306} C_VEL
LIN {X 0,Y 317.522,Z 569.609,A -85,B 0,C 180,E1 -15688.057,E2 -15688.057} C_VEL
LIN {X 0,Y 315.111,Z 557.408,A -85,B 0,C 180,E1 -15690.567,E2 -15690.567} C_VEL
LIN {X 0,Y 312.571,Z 545.729,A -85,B 0,C 180,E1 -15693.047,E2 -15693.047} C_VEL
LIN {X 0,Y 312.54,Z 545.555,A -85,B 0,C 180,E1 -15695.949,E2 -15695.949} C_VEL
LIN {X 0,Y 312.513,Z 545.553,A -85,B 0,C 180,E1 -15699.027,E2 -15699.027} C_VEL
LIN {X 0,Y 312.497,Z 545.514,A -85,B 0,C 180,E1 -15702.431,E2 -15702.431} C_VEL
LIN {X 0,Y 312.527,Z 545.55,A -85,B 0,C 180,E1 -15706.022,E2 -15706.022} C_VEL
LIN {X 0,Y 312.511,Z 545.528,A -85,B 0,C 180,E1 -15709.874,E2 -15709.874} C_VEL
LIN {X 0,Y 312.54,Z 545.554,A -85,B 0,C 180,E1 -15714.05,E2 -15714.05} C_VEL
LIN {X 0,Y 312.509,Z 545.559,A -85,B 0,C 180,E1 -15717.333,E2 -15717.333} C_VEL
LIN {X 0,Y 312.616,Z 545.752,A -85,B 0,C 180,E1 -15721.402,E2 -15721.402} C_VEL
LIN {X 0,Y 314.374,Z 553.725,A -85,B 0,C 180,E1 -15724.179,E2 -15724.179} C_VEL
LIN {X 0,Y 318.02,Z 562.559,A -85,B 0,C 180,E1 -15724.767,E2 -15724.767} C_VEL
LIN {X 0,Y 322.731,Z 575.207,A -85,B 0,C 180,E1 -15725.468,E2 -15725.468} C_VEL
LIN {X 0,Y 324.684,Z 585.818,A -85,B 0,C 180,E1 -15725.88,E2 -15725.88} C_VEL
LIN {X 0,Y 322.899,Z 659.974,A -85,B 0,C 180,E1 -15727.526,E2 -15727.526} C_VEL
LIN {X 0,Y 322.208,Z 673.377,A -85,B 0,C 180,E1 -15728.065,E2 -15728.065} C_VEL
LIN {X 0,Y 321.281,Z 686.139,A -85,B 0,C 180,E1 -15728.841,E2 -15728.841} C_VEL
LIN {X 0,Y 320.091,Z 697.462,A -85,B 0,C 180,E1 -15729.768,E2 -15729.768} C_VEL
LIN {X 0,Y 318.646,Z 709.109,A -85,B 0,C 180,E1 -15731.014,E2 -15731.014} C_VEL
LIN {X 0,Y 317.372,Z 719.423,A -85,B 0,C 180,E1 -15732.417,E2 -15732.417} C_VEL
LIN {X 0,Y 316.084,Z 728.098,A -85,B 0,C 180,E1 -15733.862,E2 -15733.862} C_VEL
LIN {X 0,Y 314.813,Z 735.965,A -85,B 0,C 180,E1 -15735.453,E2 -15735.453} C_VEL
LIN {X 0,Y 313.561,Z 743.65,A -85,B 0,C 180,E1 -15737.376,E2 -15737.376} C_VEL
LIN {X 0,Y 312.397,Z 750.707,A -85,B 0,C 180,E1 -15739.631,E2 -15739.631} C_VEL
LIN {X 0,Y 311.698,Z 755.403,A -85,B 0,C 180,E1 -15741.571,E2 -15741.571} C_VEL
LIN {X 0,Y 311.268,Z 758.991,A -85,B 0,C 180,E1 -15743.517,E2 -15743.517} C_VEL
LIN {X 0,Y 311.09,Z 760.844,A -85,B 0,C 180,E1 -15744.814,E2 -15744.814} C_VEL
LIN {X 0,Y 310.928,Z 762.241,A -85,B 0,C 180,E1 -15746.111,E2 -15746.111} C_VEL
LIN {X 0,Y 310.701,Z 763.849,A -85,B 0,C 180,E1 -15748.703,E2 -15748.703} C_VEL
LIN {X 0,Y 310.698,Z 764.081,A -85,B 0,C 180,E1 -15749.999,E2 -15749.999} C_VEL
LIN {X 0,Y 310.7,Z 763.891,A -85,B 0,C 180,E1 -15751.295,E2 -15751.295} C_VEL
LIN {X 0,Y 310.923,Z 762.339,A -85,B 0,C 180,E1 -15753.887,E2 -15753.887} C_VEL
LIN {X 0,Y 311.084,Z 760.984,A -85,B 0,C 180,E1 -15755.184,E2 -15755.184} C_VEL
LIN {X 0,Y 311.392,Z 758.118,A -85,B 0,C 180,E1 -15757.129,E2 -15757.129} C_VEL
LIN {X 0,Y 311.868,Z 754.229,A -85,B 0,C 180,E1 -15759.075,E2 -15759.075} C_VEL
LIN {X 0,Y 312.703,Z 749.213,A -85,B 0,C 180,E1 -15761.012,E2 -15761.012} C_VEL
LIN {X 0,Y 313.678,Z 742.898,A -85,B 0,C 180,E1 -15762.946,E2 -15762.946} C_VEL
LIN {X 0,Y 314.945,Z 734.989,A -85,B 0,C 180,E1 -15764.868,E2 -15764.868} C_VEL
LIN {X 0,Y 316.624,Z 725.147,A -85,B 0,C 180,E1 -15766.77,E2 -15766.77} C_VEL
LIN {X 0,Y 317.97,Z 714.82,A -85,B 0,C 180,E1 -15768.357,E2 -15768.357} C_VEL
LIN {X 0,Y 319.268,Z 704.591,A -85,B 0,C 180,E1 -15769.614,E2 -15769.614} C_VEL
LIN {X 0,Y 320.6,Z 693.384,A -85,B 0,C 180,E1 -15770.699,E2 -15770.699} C_VEL
LIN {X 0,Y 321.779,Z 680.745,A -85,B 0,C 180,E1 -15771.626,E2 -15771.626} C_VEL
LIN {X 0,Y 322.587,Z 668.083,A -85,B 0,C 180,E1 -15772.284,E2 -15772.284} C_VEL
LIN {X 0,Y 323.172,Z 655.046,A -85,B 0,C 180,E1 -15772.705,E2 -15772.705} C_VEL
LIN {X 0,Y 324.642,Z 584.643,A -85,B 0,C 180,E1 -15774.263,E2 -15774.263} C_VEL
LIN {X 0,Y 322.247,Z 573.448,A -85,B 0,C 180,E1 -15774.726,E2 -15774.726} C_VEL
LIN {X 0,Y 316.197,Z 558.365,A -85,B 0,C 180,E1 -15775.608,E2 -15775.608} C_VEL
LIN {X 0,Y 314.183,Z 555.434,A -85,B 0,C 180,E1 -15775.934,E2 -15775.934} C_VEL
LIN {X 0,Y 311.807,Z 553.355,A -85,B 0,C 180,E1 -15776.4,E2 -15776.4} C_VEL
LIN {X 0,Y 308.75,Z 551.486,A -85,B 0,C 180,E1 -15777.169,E2 -15777.169} C_VEL
LIN {X 0,Y 306.482,Z 549.605,A -85,B 0,C 180,E1 -15778.055,E2 -15778.055} C_VEL
LIN {X 0,Y 305.932,Z 548.426,A -85,B 0,C 180,E1 -15778.518,E2 -15778.518} C_VEL
LIN {X 0,Y 305.502,Z 546.428,A -85,B 0,C 180,E1 -15779.383,E2 -15779.383} C_VEL
LIN {X 0,Y 305.463,Z 546.432,A -85,B 0,C 180,E1 -15783.515,E2 -15783.515} C_VEL
LIN {X 0,Y 305.499,Z 546.425,A -85,B 0,C 180,E1 -15786.734,E2 -15786.734} C_VEL
LIN {X 0,Y 305.452,Z 546.427,A -85,B 0,C 180,E1 -15790.599,E2 -15790.599} C_VEL
LIN {X 0,Y 305.423,Z 546.43,A -85,B 0,C 180,E1 -15793.654,E2 -15793.654} C_VEL
LIN {X 0,Y 305.482,Z 546.432,A -85,B 0,C 180,E1 -15797.407,E2 -15797.407} C_VEL
LIN {X 0,Y 305.504,Z 546.404,A -85,B 0,C 180,E1 -15801.601,E2 -15801.601} C_VEL
LIN {X 0,Y 305.46,Z 546.435,A -85,B 0,C 180,E1 -15804.886,E2 -15804.886} C_VEL
LIN {X 0,Y 305.447,Z 546.433,A -85,B 0,C 180,E1 -15808.354,E2 -15808.354} C_VEL
LIN {X 0,Y 305.515,Z 546.426,A -85,B 0,C 180,E1 -15811.113,E2 -15811.113} C_VEL
LIN {X 0,Y 305.565,Z 546.421,A -85,B 0,C 180,E1 -15814.087,E2 -15814.087} C_VEL
LIN {X 0,Y 305.494,Z 546.421,A -85,B 0,C 180,E1 -15818.402,E2 -15818.402} C_VEL
LIN {X 0,Y 305.583,Z 546.42,A -85,B 0,C 180,E1 -15821.217,E2 -15821.217} C_VEL
LIN {X 0,Y 305.641,Z 546.405,A -85,B 0,C 180,E1 -15825.348,E2 -15825.348} C_VEL
LIN {X 0,Y 305.631,Z 546.402,A -85,B 0,C 180,E1 -15829.399,E2 -15829.399} C_VEL
LIN {X 0,Y 305.806,Z 546.391,A -85,B 0,C 180,E1 -15832.074,E2 -15832.074} C_VEL
LIN {X 0,Y 305.683,Z 546.405,A -85,B 0,C 180,E1 -15834.723,E2 -15834.723} C_VEL
LIN {X 0,Y 305.952,Z 546.368,A -85,B 0,C 180,E1 -15838.684,E2 -15838.684} C_VEL
LIN {X 0,Y 305.952,Z 546.374,A -85,B 0,C 180,E1 -15841.316,E2 -15841.316} C_VEL
LIN {X 0,Y 305.847,Z 546.385,A -85,B 0,C 180,E1 -15846.597,E2 -15846.597} C_VEL
LIN {X 0,Y 305.728,Z 546.392,A -85,B 0,C 180,E1 -15849.26,E2 -15849.26} C_VEL
LIN {X 0,Y 305.584,Z 546.42,A -85,B 0,C 180,E1 -15853.296,E2 -15853.296} C_VEL
LIN {X 0,Y 305.586,Z 546.407,A -85,B 0,C 180,E1 -15856.02,E2 -15856.02} C_VEL
LIN {X 0,Y 305.574,Z 546.424,A -85,B 0,C 180,E1 -15859.448,E2 -15859.448} C_VEL
LIN {X 0,Y 305.484,Z 546.427,A -85,B 0,C 180,E1 -15863.042,E2 -15863.042} C_VEL
LIN {X 0,Y 305.519,Z 546.419,A -85,B 0,C 180,E1 -15866.219,E2 -15866.219} C_VEL
LIN {X 0,Y 305.481,Z 546.433,A -85,B 0,C 180,E1 -15869.048,E2 -15869.048} C_VEL
LIN {X 0,Y 305.436,Z 546.436,A -85,B 0,C 180,E1 -15871.953,E2 -15871.953} C_VEL
LIN {X 0,Y 305.456,Z 546.422,A -85,B 0,C 180,E1 -15875.114,E2 -15875.114} C_VEL
LIN {X 0,Y 305.444,Z 546.433,A -85,B 0,C 180,E1 -15878.53,E2 -15878.53} C_VEL
LIN {X 0,Y 305.48,Z 546.416,A -85,B 0,C 180,E1 -15882.593,E2 -15882.593} C_VEL
LIN {X 0,Y 305.488,Z 546.423,A -85,B 0,C 180,E1 -15886.358,E2 -15886.358} C_VEL
LIN {X 0,Y 305.495,Z 546.425,A -85,B 0,C 180,E1 -15889.9,E2 -15889.9} C_VEL
LIN {X 0,Y 305.497,Z 546.41,A -85,B 0,C 180,E1 -15893.628,E2 -15893.628} C_VEL
LIN {X 0,Y 305.507,Z 546.515,A -85,B 0,C 180,E1 -15896.35,E2 -15896.35} C_VEL
LIN {X 0,Y 307.874,Z 556.829,A -85,B 0,C 180,E1 -15899.856,E2 -15899.856} C_VEL
LIN {X 0,Y 309.89,Z 566.829,A -85,B 0,C 180,E1 -15903.028,E2 -15903.028} C_VEL
LIN {X 0,Y 310.333,Z 569.418,A -85,B 0,C 180,E1 -15903.745,E2 -15903.745} C_VEL
LIN {X 0,Y 311.743,Z 574.792,A -85,B 0,C 180,E1 -15904.048,E2 -15904.048} C_VEL
LIN {X 0,Y 316.932,Z 605.168,A -85,B 0,C 180,E1 -15905.243,E2 -15905.243} C_VEL
LIN {X 0,Y 317.727,Z 610.849,A -85,B 0,C 180,E1 -15905.447,E2 -15905.447} C_VEL
LIN {X 0,Y 316.12,Z 677.692,A -85,B 0,C 180,E1 -15906.976,E2 -15906.976} C_VEL
LIN {X 0,Y 315.137,Z 691.617,A -85,B 0,C 180,E1 -15907.549,E2 -15907.549} C_VEL
LIN {X 0,Y 314.043,Z 704.083,A -85,B 0,C 180,E1 -15908.332,E2 -15908.332} C_VEL
LIN {X 0,Y 312.72,Z 715.203,A -85,B 0,C 180,E1 -15909.272,E2 -15909.272} C_VEL
LIN {X 0,Y 311.15,Z 726.779,A -85,B 0,C 180,E1 -15910.541,E2 -15910.541} C_VEL
LIN {X 0,Y 309.562,Z 737.203,A -85,B 0,C 180,E1 -15911.983,E2 -15911.983} C_VEL
LIN {X 0,Y 308.187,Z 746.737,A -85,B 0,C 180,E1 -15913.64,E2 -15913.64} C_VEL
